	T_ExchgParam.T_StationCommon.xOnlineValueModified_St1:=fbCompareProfileProcessValue.xProcessValueModified;
END_ACTION
ACTION ResetVisu:
(* waiting for reset *)
	RisingEdgeReset(CLK:=T_Visu.T_CtrleVisu.xReset);
	IF RisingEdgeReset.Q THEN
		(* call functionblock init. *)
		fbQvisInitPage(	T_Visu:=T_Visu);
		T_Visu.T_CtrleVisu.xDone:=FALSE;
		T_Visu.T_CtrleVisu.iFunction:=0;
		T_Visu.T_CtrleVisu.xErr:=FALSE;
		T_Visu.T_CtrleVisu.udiErrorID:=0;
		T_Visu.T_PlcParam.dwSetNewPage:=0;
		T_Visu.T_PlcParam.dwActualPage:=0;
		T_Visu.T_PlcParam.dwPreviousPage:=0;
		T_ExchgParam.T_Visu.iQVisActivNewPage:=0;
		T_ExchgParam.T_TeachIn.iSetup_AxisSel:=1;
		T_ExchgParam.T_StationCommon.xBlockSelectAutoMode:=FALSE;
		InitSavePages;
		awSaveStateTaskBar[0]:=awSaveStateTaskBar[1]:=awSaveStateTaskBar[2]:=awSaveStateTaskBar[3]:=awSaveStateTaskBar[4]:=1;
		iSaveSetupMode:=1;
		(* Activ reset structure control action *)
		T_Visu.T_CtrleAction.xReset:=TRUE;
		(* Activ reset structure control process *)
		T_Visu.T_CtrleProcess.xReset:=TRUE;
		RisingEdgeReseTProcess(CLK:=FALSE);
		(* active confirmation *)
		xConfirmResetFB:=TRUE;
		(* exit function bloc *)
		RETURN;
	ELSE
		IF xConfirmResetFB THEN
			(* confirm reset FB *)
			T_Visu.T_CtrleVisu.xDone:=TRUE;
			T_Visu.T_CtrleVisu.xErr:=FALSE;
			T_Visu.T_CtrleVisu.udiErrorID:=0;
			(* reset variable *)
			xConfirmResetFB:=FALSE;
			(* activ research if Qvis is activ *)
			xQvisActiv:=TRUE;
			T_Visu.T_CtrleVisu.xQvis:=FALSE;
			dwInCount_QVisCmd:=T_CtrleQVis.dwInCount;
		END_IF
	END_IF;
END_ACTION
ACTION UserLevel:
	RisingEdgeCheckPasswordPage(CLK:=(T_Visu.T_PlcParam.dwActualPage = gT_PageNumber.iAutoMode_UserLevel));
	IF RisingEdgeCheckPasswordPage.Q OR xChangeRandomValue THEN
		xChangeRandomValue:=FALSE;
		(* Der Counter respektive Random muss 9 Stellig sein welches aus dem Zyklusticker der CPU ausgelesen wird *)
		fbGetCpuAccount;
		FBPassword_SystemLevel(	dwCounterHI:= fbGetCpuAccount.cpuCntHiDW,
								dwCounterLOW:=fbGetCpuAccount.cpuCntLoDW);
		T_ExchgParam.T_Visu.T_Level.diRandom:=FBPassword_SystemLevel.diRandom;
	END_IF;
(* Monitor password divers level *)
	(* set Standard Level *)
	RisingEdgeStandardLevel(CLK:=(T_ExchgParam.T_Visu.T_Level.iActLevel = 0));
	IF RisingEdgeStandardLevel.Q THEN
		xChangeRandomValue:=TRUE;
		T_ExchgParam.T_Visu.T_Message.iState:=31;			(* Info: Sie sind nun als Standard angemeldet *)
	END_IF;
	(* set Operator Level *)
	IF T_ExchgParam.T_Visu.T_Level.diPwOperator <> -1 THEN
		IF T_ExchgParam.T_Visu.T_Level.diPwOperator = T_ExchgParam.T_Visu.T_Level.diPwOperatorSaved THEN
		(* pw correct *)
			T_ExchgParam.T_Visu.T_Level.iActLevel:=1;
			T_ExchgParam.T_Visu.T_Message.iState:=1;			(* Info: Sie sind nun als Operator angemeldet *)
		(* wrong pw *)
		ELSE 	T_ExchgParam.T_Visu.T_Message.iState:=204;	(* Warnung: Falsches Operator Passwort *) END_IF
		T_ExchgParam.T_Visu.T_Level.diPwOperator:=-1;
		xChangeRandomValue:=TRUE;
	END_IF;
	(* set system level *)
	IF T_ExchgParam.T_Visu.T_Level.diPwSystem <> -1 THEN
		IF T_ExchgParam.T_Visu.T_Level.diPwSystem = FBPassword_SystemLevel.diPwSystem THEN
		(* pw correct *)
			T_ExchgParam.T_Visu.T_Level.iActLevel:=2;
			T_ExchgParam.T_Visu.T_Message.iState:=2;			(* Info: Sie sind nun als System angemeldet *)
		(* wrong pw *)
		ELSE 	T_ExchgParam.T_Visu.T_Message.iState:=205; 		(* Warnung: Falsches System Passwort *) END_IF
		T_ExchgParam.T_Visu.T_Level.diPwSystem:=-1;
		xChangeRandomValue:=TRUE;
	END_IF

	IF (T_ExchgParam.T_Visu.T_Level.iActLevel > 1) THEN
		T_ExchgParam.T_StationCommon.xSystemLevelActive:=TRUE;
	ELSE
		T_ExchgParam.T_StationCommon.xSystemLevelActive:=FALSE;
	END_IF;
END_ACTION
ACTION VisuFunction_Axis:
	xTmp:=	xAxisStop OR xAxisStopAll OR xAxisTogglePower OR
			xAxisReset OR xAxisMoveContinous OR xAxisMoveAbsolut OR
			xAxisMoveRelative OR xAxisTeachPosition;

	T_ExchgParam.T_TeachIn.xDisableAxisSelectButton:=xTmp;	(* Auswahl der Achsen muss gesperrt werden im Fall einer Aktiven VisuFunktion für Achsen *)

	IF IxJoystick_X_Plus THEN
		T_ExchgParam.T_TeachIn.xJogInc_Common_Setup_Axis:=TRUE;
		T_ExchgParam.T_Visu.T_Message.iState:=35;	(* Info: Achsen auf Jog Bewegung gesetzt ! *)
	END_IF;
	IF IxJoystick_X_Minus THEN
		T_ExchgParam.T_TeachIn.xJogInc_Common_Setup_Axis:=FALSE;
		T_ExchgParam.T_Visu.T_Message.iState:=34;	(* Info: Achsen auf Ink Bewegung gesetzt ! *)
	END_IF;

(* Bewegung einer Achse stoppen *)
	IF xAxisStop THEN
		(* Step stop axis *)
		CASE iStepAction OF
		(* check Ressource *)
		1:	xTmp:=	TRUE;
			IF xTmp THEN
				(* next Step *)
				iStepAction :=10;
				xStepActionDone:=FALSE;
			(* activ error *)
			ELSE
				iStepAction:=95;
			END_IF
			xAxisMoveContinous:=FALSE;
		(* stop axis *)
		10:	ptrTCommonAxis^.T_CtrleSingle.iFunction:=5;
			ptrTCommonAxis^.T_CtrleSingle.xExecute:=TRUE;
			(* next step *)
			iStepAction:=20;
			xStepActionDone:=FALSE;
		(* waiting stop confirmation *)
		20:	IF NOT(xStepActionDone) THEN
			(* release execution *)
				ptrTCommonAxis^.T_CtrleSingle.xExecute:=FALSE;
				(* confirm step *)
				xStepActionDone:=TRUE;
			ELSE
				IF ptrTCommonAxis^.T_CtrleSingle.xDone THEN
				(* next step *)
					iStepAction:=90;
					xStepActionDone:=FALSE;
					T_ExchgParam.T_Visu.T_Message.iState:=277;	(* Warnung: Achse wurde gestoppt ! *)
				END_IF
			END_IF
		(* action done *)
		90:	T_Visu.T_CtrleAction.xDone:=TRUE;
			T_Visu.T_CtrleAction.xNotReady:=FALSE;
			T_Visu.T_CtrleAction.xErr:=FALSE;
			T_Visu.T_CtrleAction.udiErrorID:=0;
			xAxisStop:=FALSE;
		(* axis not ready *)
		95:	TimerNotReady(IN:=TRUE);
			xAxisStop:=FALSE;
		END_CASE
	END_IF;

(* Bewegung aller Achse stoppen *)
	IF xAxisStopAll THEN
		(* Step stop axis *)
		CASE iStepAction OF
		(* check Ressource *)
		1:	xTmp:=	TRUE;
			IF xTmp THEN
				(* next Step *)
				iStepAction :=10;
				xStepActionDone:=FALSE;
			(* activ error *)
			ELSE
				iStepAction:=95;
			END_IF
			xAxisMoveContinous:=FALSE;
		(* stop axis *)
		10:	IF xAxisStopAll THEN
				ptrTAxisZ_St1^.T_CtrleSingle.iFunction:=5;
				ptrTAxisZ_St1^.T_CtrleSingle.xExecute:=TRUE;
				ptrTAxisS_St1^.T_CtrleSingle.iFunction:=5;
				ptrTAxisS_St1^.T_CtrleSingle.xExecute:=TRUE;
			END_IF;
			(* next step *)
			iStepAction:=20;
			xStepActionDone:=FALSE;
		(* waiting stop confirmation *)
		20:	IF NOT(xStepActionDone) THEN
			(* release execution *)
				(* confirm step *)
				xStepActionDone:=TRUE;
			ELSE
				IF ptrTAxisZ_St1^.T_CtrleSingle.xDone AND ptrTAxisS_St1^.T_CtrleSingle.xDone THEN
				(* next step *)
					iStepAction:=90;
					xStepActionDone:=FALSE;
					T_ExchgParam.T_Visu.T_Message.iState:=277;	(* Warnung: Achse wurde gestoppt ! *)
				END_IF
			END_IF
		(* action done *)
		90:	T_Visu.T_CtrleAction.xDone:=TRUE;
			T_Visu.T_CtrleAction.xNotReady:=FALSE;
			T_Visu.T_CtrleAction.xErr:=FALSE;
			T_Visu.T_CtrleAction.udiErrorID:=0;
			xAxisStopAll:=FALSE;
		(* axis not ready *)
		95:	TimerNotReady(IN:=TRUE);
			xAxisStopAll:=FALSE;
		END_CASE
	END_IF;

(* Achsen Drehmoment Ein/Aus Toggeln *)
	IF xAxisTogglePower THEN
		(* Step toogle axis power *)
		CASE iStepAction OF
		(* check axis *)
		1:	xTmp:=	ptrTCommonAxis^.T_CtrleSingle.xDone
					AND ptrTCommonAxis^.T_CtrleSingle.xNotMoving
					AND NOT(ptrTCommonAxis^.T_CtrleSingle.xErr)
					AND NOT(ptrTCommonAxis^.T_CtrleSingle.xExecute);
			IF xTmp THEN
				iStepAction:=10;
			ELSE
				iStepAction:=95;
			END_IF
		(* activ function axis *)
		10:	IF ptrTCommonAxis^.T_CtrleSingle.xPower THEN ptrTCommonAxis^.T_CtrleSingle.iFunction:=4;
				ELSE ptrTCommonAxis^.T_CtrleSingle.iFunction:=3; END_IF
			ptrTCommonAxis^.T_CtrleSingle.xExecute:=TRUE;
			(* next step *)
			iStepAction:=20;
			xStepActionDone:=FALSE;
		(* confirm execution *)
		20:	IF NOT(xStepActionDone) THEN
			(* confirm execution *)
				ptrTCommonAxis^.T_CtrleSingle.xExecute:=FALSE;
				xStepActionDone:=TRUE;
			ELSE
				IF ptrTCommonAxis^.T_CtrleSingle.xDone THEN
					IF (ptrTCommonAxis^.T_CtrleSingle.iFunction = 3) THEN
						T_ExchgParam.T_Visu.T_Message.iState:=7;	(* Info: Achsenstrom EIN ! *)
					ELSE
						T_ExchgParam.T_Visu.T_Message.iState:=8;	(* Info: Achsenstrom AUS ! *)
					END_IF
				(* confirm action next step *)
					iStepAction:=90;
					xStepActionDone:=FALSE;
				END_IF
			END_IF
		(* action done *)
		90:	T_Visu.T_CtrleAction.xDone:=TRUE;
			T_Visu.T_CtrleAction.xNotReady:=FALSE;
			T_Visu.T_CtrleAction.xErr:=FALSE;
			T_Visu.T_CtrleAction.udiErrorID:=0;
			xAxisTogglePower:=FALSE;
		(* Axis not ready *)
		95:	TimerNotReady(IN:=TRUE);
			xAxisTogglePower:=FALSE;
		END_CASE
	END_IF

(* Achse Resetten *)
	IF xAxisReset THEN
		(* Step reset axis *)
		CASE iStepAction OF
		(* check axis *)
		1:	xTmp:=	NOT(ptrTCommonAxis^.T_CtrleSingle.xExecute);
			IF xTmp THEN
				iStepAction:=10;
			ELSE iStepAction:=95;
			END_IF
		(* activ function axis *)
		10:	ptrTCommonAxis^.T_CtrleSingle.iFunction:=1;
			ptrTCommonAxis^.T_CtrleSingle.xExecute:=TRUE;
			(* next step *)
			iStepAction:=20;
			xStepActionDone:=FALSE;
		(* confirm execution *)
		20:	IF NOT(xStepActionDone) THEN
			(* confirm execution *)
				ptrTCommonAxis^.T_CtrleSingle.xExecute:=FALSE;
				xStepActionDone:=TRUE;
			ELSE
				IF ptrTCommonAxis^.T_CtrleSingle.xDone THEN
					T_ExchgParam.T_Visu.T_Message.iState:=9;	(* Info: Achse erfolgreich Zurückgesetzt ! *)
				(* confirm action next step *)
					iStepAction:=90;
					xStepActionDone:=FALSE;
				END_IF
			END_IF
		(* action done *)
		90:	T_Visu.T_CtrleAction.xDone:=TRUE;
			T_Visu.T_CtrleAction.xNotReady:=FALSE;
			T_Visu.T_CtrleAction.xErr:=FALSE;
			T_Visu.T_CtrleAction.udiErrorID:=0;
			xAxisReset:=FALSE;
		(* Axis not ready *)
		95:	TimerNotReady(IN:=TRUE);
			xAxisReset:=FALSE;
		END_CASE
	END_IF

(* Achse Geschwindigkeitsmodus *)
	IF xAxisMoveContinous THEN
		(* Step move continuous velocity *)
		CASE iStepAction OF
		(* check axis *)
		1:	xTmp:=	ptrTCommonAxisActive^.T_CtrleSingle.xDone
					AND ptrTCommonAxisActive^.T_CtrleSingle.xReady
					AND ptrTCommonAxisActive^.T_CtrleSingle.xNotMoving
					AND NOT(ptrTCommonAxisActive^.T_CtrleSingle.xErr)
					AND NOT(ptrTCommonAxisActive^.T_CtrleSingle.xExecute);
			IF (ptrTCommonAxisActive^.T_CtrleSingle.lrVelocity = 0) THEN
				(* Geschwindigkeit darf nicht 0 sein *)
				iStepAction:=90;
				T_ExchgParam.T_Visu.T_Message.iState:=288;	(* Warnung: Geschwindigkeit muss grösser als 0 sein ! *)
				RETURN;
			END_IF;
			IF xTmp THEN
				iStepAction:=10;
			ELSE
				iStepAction:=95;
			END_IF
		(* activ function axis *)
		10:	ptrTCommonAxisActive^.T_CtrleSingle.iFunction:=6;
			ptrTCommonAxisActive^.T_CtrleSingle.xExecute:=TRUE;
			ptrTCommonAxisActive^.T_CtrleSingle.lrAcceleration:=TCommonTeachParameter.rAcceleration;
			ptrTCommonAxisActive^.T_CtrleSingle.lrDecceleration:=TCommonTeachParameter.rDeceleration;
			ptrTCommonAxisActive^.T_CtrleSingle.lrJerk:=TCommonTeachParameter.rJerk;
			(* next step *)
			iStepAction:=20;
			xStepActionDone:=FALSE;
			T_ExchgParam.T_Visu.T_Message.iState:=14;	(* Info: Achsenbewegung gestartet ! *)
		(* confirm execution *)
		20:	IF NOT(xStepActionDone) THEN
			(* confirm execution *)
				ptrTCommonAxisActive^.T_CtrleSingle.xExecute:=FALSE;
				xStepActionDone:=TRUE;
			ELSE
				IF ptrTCommonAxisActive^.T_CtrleSingle.xDone THEN
					xStepActionDone:=FALSE;
					(* confirm action next step *)
					iStepAction:=90;
				END_IF
			END_IF
		(* action done *)
		90:	T_Visu.T_CtrleAction.xDone:=TRUE;
			T_Visu.T_CtrleAction.xNotReady:=FALSE;
			T_Visu.T_CtrleAction.xErr:=FALSE;
			T_Visu.T_CtrleAction.udiErrorID:=0;
			xAxisMoveContinous:=FALSE;
		(* axis not ready *)
		95:	TimerNotReady(IN:=TRUE);
			xAxisMoveContinous:=FALSE;
		END_CASE
	END_IF

(* Achse Absolute Positionsbewegung *)
	IF xAxisMoveAbsolut THEN
		(* Step move abs position *)
		CASE iStepAction OF
		(* check axis *)
		1:	xTmp:=	ptrTCommonAxis^.T_CtrleSingle.xDone
					AND ptrTCommonAxis^.T_CtrleSingle.xReady
					AND ptrTCommonAxis^.T_CtrleSingle.xNotMoving
					AND NOT(ptrTCommonAxis^.T_CtrleSingle.xErr)
					AND NOT(ptrTCommonAxis^.T_CtrleSingle.xExecute);
			IF xTmp THEN
				IF NOT(ptrTCommonAxis^.T_CtrleSingle.xRef) THEN
					T_ExchgParam.T_Visu.T_Message.iState:=206;	(* Warnung: Ausgewählte Achse ist nicht referenziert ! *)
					iStepAction:=90;
				ELSE
					iStepAction:=10;
				END_IF
			ELSE
				iStepAction:=95;
			END_IF;
		(* waiting confirmation *)
		10:	(* init. acc/dec/jerk *)
			ptrTCommonAxis^.T_CtrleSingle.lrAcceleration:=TCommonTeachParameter.rAcceleration;
			ptrTCommonAxis^.T_CtrleSingle.lrDecceleration:=TCommonTeachParameter.rDeceleration;
			ptrTCommonAxis^.T_CtrleSingle.lrJerk:=TCommonTeachParameter.rJerk;
			ptrTCommonAxis^.T_CtrleSingle.lrVelocity:=TCommonTeachParameter.rPositionSpeed;
			ptrTCommonAxis^.T_CtrleSingle.lrPosition:=TCommonTeachParameter.rRefPosition;
			ptrTCommonAxis^.T_CtrleSingle.xExecute:=TRUE;
			ptrTCommonAxis^.T_CtrleSingle.iFunction:=7;
			iStepAction:=20;
			xStepActionDone:=FALSE;
			IF NOT(xAxisLimitSwitchActive) THEN
				T_ExchgParam.T_Visu.T_Message.iState:=15;	(* Info: Achse fährt auf ausgewählte Position ! *)
			END_IF;
			gxAxisAbsolutMovementActive:=TRUE;	(* Damit die Achsen mit dem Override gesetzt werden bezüglich der Absoluten Bewegung *)
		(* confirm execution *)
		20:	IF NOT(xStepActionDone) THEN
			(* confirm execution *)
				ptrTCommonAxis^.T_CtrleSingle.xExecute:=FALSE;
				xStepActionDone:=TRUE;
			ELSE
				IF ptrTCommonAxis^.T_CtrleSingle.xDone THEN
					xStepActionDone:=FALSE;
					(* confirm action next step *)
					iStepAction:=90;
					IF NOT(xAxisLimitSwitchActive) THEN
						T_ExchgParam.T_Visu.T_Message.iState:=16;	(* Info: Achsenposition erreicht ! *)
					END_IF;
				END_IF
			END_IF;
		(* action done *)
		90:	T_Visu.T_CtrleAction.xDone:=TRUE;
			T_Visu.T_CtrleAction.xNotReady:=FALSE;
			T_Visu.T_CtrleAction.xErr:=FALSE;
			T_Visu.T_CtrleAction.udiErrorID:=0;
			xAxisMoveAbsolut:=FALSE;
		(* axis not ready *)
		95:	TimerNotReady(IN:=TRUE);
			xAxisMoveAbsolut:=FALSE;
		END_CASE
	END_IF

(* Achse Relative Positionsbewegung *)
	IF xAxisMoveRelative THEN
		(* Step move abs position *)
		CASE iStepAction OF
		(* check axis *)
		1:	xTmp:=	ptrTCommonAxisActive^.T_CtrleSingle.xDone
					AND ptrTCommonAxisActive^.T_CtrleSingle.xReady
					AND ptrTCommonAxisActive^.T_CtrleSingle.xNotMoving
					AND NOT(ptrTCommonAxisActive^.T_CtrleSingle.xErr)
					AND NOT(ptrTCommonAxisActive^.T_CtrleSingle.xExecute);
			IF xTmp THEN
				iStepAction:=10;
			ELSE
				iStepAction:=95;
			END_IF;
		(* Überprüfe Software Endschalter *)
		10:	IF ptrTCommonAxisActive^.T_CtrleSingle.xSWLimitSwitchPosActivated THEN
				IF ((ptrTCommonAxisActive^.T_LiveValue.lrActualPosition + ptrTCommonAxisActive^.T_CtrleSingle.lrDistance) > 0.1) THEN
					(* Überschreibe den Inkrement, damit die Achse nicht einen Fehler auswertet! Melde es dann als Softwareendschalter *)
					ptrTCommonAxisActive^.T_CtrleSingle.lrDistance:=0.09 - ptrTCommonAxisActive^.T_LiveValue.lrActualPosition;
					IF ((ptrTCommonAxisActive^.T_LiveValue.lrActualPosition + 0.01) >= 0.1) THEN
						ptrTCommonAxisActive^.T_CtrleSingle.lrDistance:=0.0;
					END_IF;
				END_IF;
			END_IF;
			iStepAction:=20;
		(* waiting confirmation *)
		20:	(* init. acc/dec/jerk *)
			ptrTCommonAxisActive^.T_CtrleSingle.lrAcceleration:=TCommonTeachParameter.rAcceleration;
			ptrTCommonAxisActive^.T_CtrleSingle.lrDecceleration:=TCommonTeachParameter.rDeceleration;
			ptrTCommonAxisActive^.T_CtrleSingle.lrJerk:=TCommonTeachParameter.rJerk;
			ptrTCommonAxisActive^.T_CtrleSingle.iFunction:=8;	(* Relative Bewegung *)
			ptrTCommonAxisActive^.T_CtrleSingle.xExecute:=TRUE;
			iStepAction:=30;
			xStepActionDone:=FALSE;
			IF NOT(xAxisLimitSwitchActive) THEN
				T_ExchgParam.T_Visu.T_Message.iState:=21;	(* Info: Achse relative Bewegung gestartet ! *)
			END_IF;
		(* confirm execution *)
		30:	IF NOT(xStepActionDone) THEN
			(* confirm execution *)
				ptrTCommonAxisActive^.T_CtrleSingle.xExecute:=FALSE;
				xStepActionDone:=TRUE;
			ELSE
				IF ptrTCommonAxisActive^.T_CtrleSingle.xDone THEN
					xStepActionDone:=FALSE;
					(* confirm action next step *)
					iStepAction:=90;
					IF NOT(xAxisLimitSwitchActive) THEN
						T_ExchgParam.T_Visu.T_Message.iState:=22;	(* Info: Achse relative Bewegung durchgeführt ! *)
					END_IF;
				END_IF
			END_IF;
		(* action done *)
		90:	T_Visu.T_CtrleAction.xDone:=TRUE;
			T_Visu.T_CtrleAction.xNotReady:=FALSE;
			T_Visu.T_CtrleAction.xErr:=FALSE;
			T_Visu.T_CtrleAction.udiErrorID:=0;
			xAxisMoveRelative:=FALSE;
		(* axis not ready *)
		95:	TimerNotReady(IN:=TRUE);
			xAxisMoveRelative:=FALSE;
		END_CASE
	END_IF

(* Z Achse auf WzWechsel Pos oder auf Z Achse auf LadePos setzen *)
	IF xZAxisMoveToToolChangePos OR xZAxisMoveToLoadPos THEN
		(* Step move abs position *)
		CASE iStepAction OF
		(* check axis *)
		1:	xTmp:=	ptrTCommonAxisActive^.T_CtrleSingle.xDone
					AND ptrTCommonAxisActive^.T_CtrleSingle.xReady
					AND ptrTCommonAxisActive^.T_CtrleSingle.xNotMoving
					AND NOT(ptrTCommonAxisActive^.T_CtrleSingle.xErr)
					AND NOT(ptrTCommonAxisActive^.T_CtrleSingle.xExecute);
			IF xTmp THEN
				IF NOT(ptrTCommonAxisActive^.T_CtrleSingle.xRef) THEN
					T_ExchgParam.T_Visu.T_Message.iState:=206;	(* Warnung: Ausgewählte Achse ist nicht referenziert ! *)
					iStepAction:=90;
				ELSE
					iStepAction:=5;
					T_ExchgParam.T_Visu.T_Message.iState:=109;	(* Aufforderung: Z Achse Position anfahren <Enter>, abbrechen <Esc> ? *)
				END_IF
			ELSE
				iStepAction:=95;
			END_IF;
		(* Set Value *)
		5:	IF RisingEdgeKeyPanel_Enter.Q THEN
				(* Display message *)
				tTimeOutAction:=T#999999s;
				iStepAction:=10;
			ELSE
				IF RisingEdgeKeyPanel_Esc.Q THEN
					iStepAction:=90;
					T_ExchgParam.T_Visu.T_Message.iState:=202;	(* Warnung: Aktion abgebrochen ! *)
				END_IF
			END_IF
			(* An other message has been displayed *)
			IF (T_ExchgParam.T_Visu.T_Message.iState<>3) AND (T_ExchgParam.T_Visu.T_Message.iState<>109) AND (T_ExchgParam.T_Visu.T_Message.iState<>202) THEN iStepAction:=90; END_IF
		(* waiting confirmation *)
		10:	(* init. acc/dec/jerk *)
			ptrTCommonAxisActive^.T_CtrleSingle.xExecute:=TRUE;
			ptrTCommonAxisActive^.T_CtrleSingle.iFunction:=7;
			ptrTCommonAxisActive^.T_CtrleSingle.lrPosition:=rZAxisSelectPosition;
			iStepAction:=20;
			xStepActionDone:=FALSE;
			IF NOT(xAxisLimitSwitchActive) THEN
				T_ExchgParam.T_Visu.T_Message.iState:=15;	(* Info: Achse fährt auf ausgewählte Position ! *)
			END_IF;
			gxAxisAbsolutMovementActive:=TRUE;	(* Damit die Achsen mit dem Override gesetzt werden bezüglich der Absoluten Bewegung *)
		(* confirm execution *)
		20:	IF NOT(xStepActionDone) THEN
			(* confirm execution *)
				ptrTCommonAxisActive^.T_CtrleSingle.xExecute:=FALSE;
				xStepActionDone:=TRUE;
			ELSE
				IF ptrTCommonAxisActive^.T_CtrleSingle.xDone THEN
					xStepActionDone:=FALSE;
					(* confirm action next step *)
					iStepAction:=90;
					IF NOT(xAxisLimitSwitchActive) THEN
						T_ExchgParam.T_Visu.T_Message.iState:=16;	(* Info: Achsenposition erreicht ! *)
					END_IF;
				END_IF
			END_IF;
		(* action done *)
		90:	T_Visu.T_CtrleAction.xDone:=TRUE;
			T_Visu.T_CtrleAction.xNotReady:=FALSE;
			T_Visu.T_CtrleAction.xErr:=FALSE;
			T_Visu.T_CtrleAction.udiErrorID:=0;
			xZAxisMoveToToolChangePos:=xZAxisMoveToLoadPos:=FALSE;
		(* axis not ready *)
		95:	TimerNotReady(IN:=TRUE);
			xZAxisMoveToToolChangePos:=xZAxisMoveToLoadPos:=FALSE;
		END_CASE
	END_IF

(* Meldung ausgeben, falls bei den Achse Z  Endschalter angefahren werden *)
	IF T_StartUp.T_State.xCompleted THEN
		IF ptrTAxisZ_St1^.T_CtrleSingle.xHWLimitNeg THEN
			T_ExchgParam.T_Visu.T_Message.iState:=209;	(* Warnung: Z-Achse negativer HW Endschalter angefahren ! *)
		END_IF;
		IF ptrTAxisZ_St1^.T_CtrleSingle.xHWLimitPos THEN
			T_ExchgParam.T_Visu.T_Message.iState:=210;	(* Warnung: Z-Achse positiver HW Endschalter angefahren ! *)
		END_IF;
	END_IF;

	IF (T_ExchgParam.T_Visu.T_Message.iState >= 209) AND (T_ExchgParam.T_Visu.T_Message.iState <= 210) THEN
		xAxisLimitSwitchActive:=TRUE;
	ELSE
		xAxisLimitSwitchActive:=FALSE;
	END_IF;

(* Löschen der berechnete Wert für Wippe des Drehmoment Detection *)
IF xResetRockerValue THEN
	grRockerQualityMin:=grRockerQuality;
	grRockerQualityMax:=grRockerQuality;
	grRockerAmplitudeMin:=grRockerAmplitude;
	grRockerAmplitudeMax:=grRockerAmplitude;
	T_ExchgParam.T_StationCommon.rRockerQuality:=grRockerQuality:=0.0;
	T_ExchgParam.T_StationCommon.rRockerAmplitude:=grRockerAmplitude:=0.0;
	T_ExchgParam.T_StationCommon.diRockerCountHC:=gdiRockerCountHC:=0;
	T_ExchgParam.T_StationCommon.diRockerCountHCTime:=gdiRockerCountHCTime:=0;
	T_Visu.T_CtrleAction.xDone:=TRUE;
	T_Visu.T_CtrleAction.xNotReady:=FALSE;
	T_Visu.T_CtrleAction.xErr:=FALSE;
	T_Visu.T_CtrleAction.udiErrorID:=0;
	xResetRockerValue:=FALSE;
END_IF;
END_ACTION
ACTION VisuFunction_AxisTeach:
(* Achse Teach Position *)
	IF xAxisTeachPosition THEN
		CASE iStepAction OF
		(* check axis *)
		1:	xTmp:=	ptrTCommonAxis^.T_CtrleSingle.xDone
					AND ptrTCommonAxis^.T_CtrleSingle.xReady
					AND ptrTCommonAxis^.T_CtrleSingle.xNotMoving
					AND NOT(ptrTCommonAxis^.T_CtrleSingle.xErr)
					AND NOT(ptrTCommonAxis^.T_CtrleSingle.xExecute);
			xReferenceState:=ptrTCommonAxis^.T_CtrleSingle.xRef;
			IF xTmp OR gxHardwareOFF OR gxAxisOFF THEN
				IF NOT(xReferenceState) AND NOT(gxHardwareOFF) AND NOT(gxAxisOFF) THEN
					T_ExchgParam.T_Visu.T_Message.iState:=206;	(* Warnung: Ausgewählte Achse ist nicht referenziert ! *)
					iStepAction:=90;
				ELSE
					iStepAction:=2;
				END_IF
			ELSE
				iStepAction:=95;
			END_IF;
		(* Überprüfe zuerst ob die ausgewählte Position teach bar ist *)
		2:	 T_ExchgParam.T_Visu.T_Message.iState:=0;
			CASE T_ExchgParam.T_TeachIn.iSetup_AxisSel  OF
			1:	(* Z Axis *)
				IF NOT(T_NovRam.T_Parameter.T_StationWork[1].T_StProcess.xConfigActive) THEN
					IF (T_ExchgParam.T_TeachIn.arAxis[T_ExchgParam.T_TeachIn.iSetup_AxisSel].iTeachSelPos = 0) THEN
						T_ExchgParam.T_Visu.T_Message.iState:=207;			(* Warnung: Neue Position kann nicht versetzt werden ! *)
					ELSIF (T_ExchgParam.T_TeachIn.arAxis[T_ExchgParam.T_TeachIn.iSetup_AxisSel].iTeachSelPos = 6) THEN
						T_ExchgParam.T_Visu.T_Message.iState:=208;			(* Warnung: Ausgewählte Position kann nicht gespeichert werden ! *)
					END_IF;
				ELSE
					IF (T_ExchgParam.T_TeachIn.arAxis[T_ExchgParam.T_TeachIn.iSetup_AxisSel].iTeachSelPos = 0) THEN
						T_ExchgParam.T_Visu.T_Message.iState:=207;			(* Warnung: Neue Position kann nicht versetzt werden ! *)
					ELSIF (T_ExchgParam.T_TeachIn.arAxis[T_ExchgParam.T_TeachIn.iSetup_AxisSel].iTeachSelPos <= 4) THEN
						T_ExchgParam.T_Visu.T_Message.iState:=208;			(* Warnung: Ausgewählte Position kann nicht gespeichert werden ! *)
					ELSIF (T_ExchgParam.T_TeachIn.arAxis[T_ExchgParam.T_TeachIn.iSetup_AxisSel].iTeachSelPos = 6) THEN
						T_ExchgParam.T_Visu.T_Message.iState:=208;			(* Warnung: Ausgewählte Position kann nicht gespeichert werden ! *)
					END_IF;
				END_IF;
			END_CASE
			IF (T_ExchgParam.T_Visu.T_Message.iState = 0) THEN
				iStepAction:=10;
			ELSE
				(* Action has been cancelled *)
				iStepAction:=90;
			END_IF;
		(* Display message to ask for confirmation *)
		10:	T_ExchgParam.T_Visu.T_Message.iState:=103;	(* Aufforderung: Speichern bestätigen <Enter>, abbrechen <Esc> ? *)
			iStepAction:=20;
		(* waiting for key <Enter> or <Esc> *)
		20:	IF RisingEdgeKeyPanel_Enter.Q THEN
					iStepAction:=30;
			ELSIF RisingEdgeKeyPanel_Esc.Q THEN
					 iStepAction:=90;
					T_ExchgParam.T_Visu.T_Message.iState:=202;	(* Warnung: Aktion abgebrochen ! *)
			 END_IF
			(* An other message has been displayed *)
			IF (T_ExchgParam.T_Visu.T_Message.iState<>103) AND (T_ExchgParam.T_Visu.T_Message.iState<>202) THEN iStepAction:=90; END_IF
		30:	T_ExchgParam.T_Visu.T_Message.iState:=0;
			(*copy actual value to tmp variable*)
			rtmpAxisPosZ:=LREAL_TO_REAL(TStation_Work_St1.THWWorkStation.TAxisZ.T_LiveValue.lrActualPosition);
			CASE T_ExchgParam.T_TeachIn.iSetup_AxisSel  OF
			1:	(* Z Axis *)
				CASE T_ExchgParam.T_TeachIn.arAxis[T_ExchgParam.T_TeachIn.iSetup_AxisSel].iTeachSelPos OF
				(* < Z LadePos > *)
				1:	T_NovRam.T_Parameter.T_StationWork[gciStationSt1].T_StProcess.rPositionLoad:=rtmpAxisPosZ;
				(* < Z Bearb StartPos > *)
				2:	T_NovRam.T_Parameter.T_StationWork[gciStationSt1].T_StProcess.rPositionStartProc:=rtmpAxisPosZ;
				(* < Z ZentrierPos > *)
				3:	T_NovRam.T_Parameter.T_StationWork[gciStationSt1].T_StProcess.rCentringPosZ1Axis:=rtmpAxisPosZ;
				(* < Z Bearb EndPos > *)
				4:	T_NovRam.T_Parameter.T_StationWork[gciStationSt1].T_StProcess.rPositionEndProc:=rtmpAxisPosZ;
				(* < Z WzWechsel Pos > *)
				5:	T_NovRam.T_Parameter.T_StationWork[gciStationSt1].T_StProcess.rPositionToolChange:=rtmpAxisPosZ;
				(* < Z Bearb EndPos berechn. > *)
				7:	garPositionEndProcCalc[1]:=rtmpAxisPosZ;
					T_ExchgParam.T_StationCommon.rPositionEndProcCalc:=rtmpAxisPosZ;
				(* < Z Bearb EndPos Max > *)
				8:	T_NovRam.T_Parameter.T_StationWork[gciStationSt1].T_StProcess.rPositionEndProcMaxInc:=rtmpAxisPosZ;
				(* < Z ZentrierPos berechn. > *)
				9:	garCentringEndProcCalc[1]:=rtmpAxisPosZ;
					T_ExchgParam.T_StationCommon.rCentringEndProcCalc:=rtmpAxisPosZ;
				(* < Z WzZylinder Pos > *)
				10:	T_NovRam.T_Parameter.T_StationWork[gciStationSt1].T_StProcess.rZPositionCylindricalArea:=rtmpAxisPosZ;
				END_CASE;
				xUpdateStationParameter:=TRUE;
			END_CASE;
			(* Speichern der Daten in den NovRAM *)
			iStepAction:=70;
		70:	IF (garPositionEndProcCalc[1] <> T_ExchgParam.T_StationCommon.rPositionEndProcCalc) THEN
				T_ExchgParam.T_StationCommon.rPositionEndProcCalc:=garPositionEndProcCalc[1];
			END_IF;
			IF (garCentringEndProcCalc[1] <> T_ExchgParam.T_StationCommon.rCentringEndProcCalc) THEN
				T_ExchgParam.T_StationCommon.rCentringEndProcCalc:=garCentringEndProcCalc[1];
			END_IF;
			xAction_SaveNovRAM:=TRUE;
			xBlockSetNovRamAction_End:=TRUE;
			iStepActionNovRam:=1;
			iStepAction:=80;
		80:	IF NOT(xAction_SaveNovRAM) THEN
				iStepAction:=90;
				T_ExchgParam.T_Visu.T_Message.iState:=25;	(* Info: Ausgewählte Position ist nun gespeichert ! *)
			END_IF;
		(* axis not ready *)
		95:	TimerNotReady(IN:=TRUE);
			xAxisTeachPosition:=FALSE;
		(* slow/fast configuration done *)
		90:	T_Visu.T_CtrleAction.xDone:=TRUE;
			T_Visu.T_CtrleAction.xNotReady:=FALSE;
			T_Visu.T_CtrleAction.xErr:=FALSE;
			T_Visu.T_CtrleAction.udiErrorID:=0;
			xAxisTeachPosition:=FALSE;
		END_CASE
	END_IF
END_ACTION
ACTION VisuFunction_ChangePassword:
(* Ändern des Operator Passwortes *)
	IF xChangeOperatorPassword THEN
		CASE iStepAction OF
		(* Display message to ask for confirmation *)
		1:	T_ExchgParam.T_Visu.T_Level.xShow_Overlay_NewPassword:=TRUE;
			T_ExchgParam.T_Visu.T_Level.diInputOldPasword:=0;
			T_ExchgParam.T_Visu.T_Level.diInputNewPasword:=0;
			T_ExchgParam.T_Visu.T_Level.diInputRepeatPasword:=0;
			T_ExchgParam.T_Visu.T_Level.xButton_OK:=FALSE;
			T_ExchgParam.T_Visu.T_Level.xButton_Abord:=FALSE;
			iStepAction:=10;
		10:	IF T_ExchgParam.T_Visu.T_Level.xButton_OK THEN
				T_ExchgParam.T_Visu.T_Level.xButton_OK:=FALSE;
				 tTimeOutAction:=TimerAction.ET+T#3s;
				iStepAction:=20;
			END_IF;
			IF T_ExchgParam.T_Visu.T_Level.xButton_Abord THEN
				T_ExchgParam.T_Visu.T_Level.xButton_Abord:=FALSE;
				iStepAction:=90;
			END_IF;
			IF TimerAction.Q THEN iStepAction:=90; END_IF;
		(* Überprüfe Eingabe des alten Passwort *)
		20:	IF (T_ExchgParam.T_Visu.T_Level.diInputOldPasword = T_ExchgParam.T_Visu.T_Level.diPwOperatorSaved) THEN
				(* Eingabe Korrekt *)
				iStepAction:=30;
			ELSE
				T_ExchgParam.T_Visu.T_Message.iState:=214;	(* Warnung: Altes Operator Passwort falsch eingegeben ! *)
				iStepAction:=90;
			END_IF;
		(* Überprüfe Eingabe des neuen Passwort mit der Eingabe des bestätigten neuen Passwortes *)
		30:	IF (T_ExchgParam.T_Visu.T_Level.diInputNewPasword = T_ExchgParam.T_Visu.T_Level.diInputRepeatPasword) THEN
				(* Eingabe Korrekt *)
				iStepAction:=40;
			ELSE
				T_ExchgParam.T_Visu.T_Message.iState:=215;	(* Warnung: Keine Übereinstimmung der beiden neuen Operator Passwörter ! *)
				iStepAction:=90;
			END_IF;
		(* Speichern des neuen Passwortes *)
		40:	T_Password.T_Ctrle.udiSetOperatorPassword:=T_ExchgParam.T_Visu.T_Level.diInputNewPasword;
			T_Password.T_Ctrle.xExecute:=TRUE;
			T_Password.T_Ctrle.iFunction:=2;
			(* next Step *)
			iStepAction :=50;
			xStepActionDone:=FALSE;
		(* wait save confirmation *)
		50:	IF NOT(xStepActionDone) THEN
				T_Password.T_Ctrle.xExecute:=FALSE;
				(* Überschreiben des alten Passwortes *)
				T_ExchgParam.T_Visu.T_Level.diPwOperatorSaved:=T_ExchgParam.T_Visu.T_Level.diInputNewPasword;
				(* confirm Step *)
				xStepActionDone:=TRUE;
			ELSE
				IF T_Password.T_Ctrle.xDone THEN
				(* next Step *)
					iStepAction :=90;
					xStepActionDone:=FALSE;
					T_ExchgParam.T_Visu.T_Message.iState:=36;	(* Info: Neues Operator Passwort wurde gespeichert und ist Aktiv ! *)
				ELSE	IF T_Password.T_Ctrle.xErr THEN
							iStepAction:=99;
							xStepActionDone:=FALSE;
						END_IF
				END_IF
			END_IF
		(* save done *)
		90:	T_Visu.T_CtrleAction.xDone:=TRUE;
			T_Visu.T_CtrleAction.xNotReady:=FALSE;
			T_Visu.T_CtrleAction.xErr:=FALSE;
			T_Visu.T_CtrleAction.udiErrorID:=0;
			xChangeOperatorPassword:=FALSE;
			T_ExchgParam.T_Visu.T_Level.xShow_Overlay_NewPassword:=FALSE;
		(* error *)
		99:	T_Visu.T_CtrleAction.xDone:=FALSE;
			T_Visu.T_CtrleAction.xNotReady:=FALSE;
			T_Visu.T_CtrleAction.xErr:=TRUE;
			T_Visu.T_CtrleAction.udiErrorID:=16#F1000 + T_Password.T_Ctrle.iFunction;
			xChangeOperatorPassword:=FALSE;
			T_ExchgParam.T_Visu.T_Level.xShow_Overlay_NewPassword:=FALSE;
			T_Password.T_Ctrle.xReset:=TRUE;
		END_CASE
	ELSE
		T_ExchgParam.T_Visu.T_Level.xShow_Overlay_NewPassword:=FALSE;
	END_IF
END_ACTION
ACTION VisuFunction_CylinderValve:
(* Set cylinder analog value *)
	IF xCylSetServoAnalogValue THEN
		(* Step analog Wert *)
		CASE iStepAction OF
		(* check cylinder state *)
		1:	xTmp:=	ptrTCommonCylinderValve^.T_CtrleCyl.xDone
					AND NOT(ptrTCommonCylinderValve^.T_CtrleCyl.xExecute)
					AND NOT(ptrTCommonCylinderValve^.T_CtrleCyl.xErr);
			(* next step *)
			IF xTmp THEN iStepAction:=10; ELSE iStepAction:=95; END_IF
		(* activ function set analog value *)
		10:	ptrTCommonCylinderValve^.T_CtrleCyl.iFunction:=4;
			ptrTCommonCylinderValve^.T_CtrleCyl.xExecute:=TRUE;
			(* next step *)
			iStepAction:=20;
			xStepActionDone:=FALSE;
		(* wait confirmation *)
		20:	IF NOT(xStepActionDone) THEN
			(* release execution *)
				ptrTCommonCylinderValve^.T_CtrleCyl.xExecute:=FALSE;
				xStepActionDone:=TRUE;
			ELSE
				IF ptrTCommonCylinderValve^.T_CtrleCyl.xDone THEN
				(* action done *)
					iStepAction:=90;
					xStepActionDone:=FALSE;
					T_ExchgParam.T_Visu.T_Message.iState:=37;	(* Info: Kraft wurde gesetzt ! *)
				END_IF
			END_IF
		(* action done *)
		90:	T_Visu.T_CtrleAction.xDone:=TRUE;
			T_Visu.T_CtrleAction.xNotReady:=FALSE;
			T_Visu.T_CtrleAction.xErr:=FALSE;
			T_Visu.T_CtrleAction.udiErrorID:=0;
			xCylSetServoAnalogValue:=FALSE;
		(* cylinder not ready *)
		95:	TimerNotReady(IN:=TRUE);
			xCylSetServoAnalogValue:=FALSE;
		END_CASE
	END_IF;

(* Zylinder/Ventile Ein/Aus Toggeln *)
	IF xCylValveToggleOnOff THEN
		(* Step toggle Zustand *)
		CASE iStepAction OF
		(* check cylinder state *)
		1:	xTmp:=	ptrTCommonCylinderValve^.T_CtrleCyl.xDone
					AND NOT(ptrTCommonCylinderValve^.T_CtrleCyl.xExecute)
					AND NOT(ptrTCommonCylinderValve^.T_CtrleCyl.xErr);
			(* next step *)
			IF xTmp THEN iStepAction:=10; ELSE iStepAction:=95; END_IF
		(* toggle cylinder state *)
		10:	ptrTCommonCylinderValve^.T_CtrleCyl.iFunction:=51;
			ptrTCommonCylinderValve^.T_CtrleCyl.xExecute:=TRUE;
			IF (ptrTCommonCylinderValve^.iCylinderTpye = 1) THEN
				ptrTCommonCylinderValve^.T_CtrleCyl.T_Analog.rForceIn:=T_NovRAM.T_Parameter.T_StationWork[gciStationSt1].T_OnlineChange.rForceDeflection;
			END_IF;
			IF (ptrTCommonCylinderValve^.iCylinderTpye = 2) THEN
				ptrTCommonCylinderValve^.T_CtrleCyl.T_Analog.rForceIn:=T_NovRAM.T_Parameter.T_StationWork[gciStationSt1].T_OnlineChange.rTorqueLevelHC;
			END_IF;
			IF (ptrTCommonCylinderValve^.iCylinderTpye = 3) THEN
				ptrTCommonCylinderValve^.T_CtrleCyl.T_Analog.rForceIn:=T_NovRAM.T_Parameter.T_StationWork[gciStationSt1].T_StProcess.rTorqueLevel_Overload;
				TStation_Work_St1.THWWorkStation.TCylToolTorqueHC.T_CtrleCyl.T_Analog.rForceIn:=T_NovRAM.T_Parameter.T_StationWork[gciStationSt1].T_OnlineChange.rTorqueLevelHC;
			END_IF;
			(* next step *)
			iStepAction:=20;
			xStepActionDone:=FALSE;
		(* wait confirmation *)
		20:	IF NOT(xStepActionDone) THEN
			(* release execution *)
				ptrTCommonCylinderValve^.T_CtrleCyl.xExecute:=FALSE;
				xStepActionDone:=TRUE;
			ELSE
				IF ptrTCommonCylinderValve^.T_CtrleCyl.xDone THEN
				(* action done *)
					iStepAction:=90;
					xStepActionDone:=FALSE;
					T_ExchgParam.T_Visu.T_Message.iState:=38;	(* Info: Zustand des Zylinderausganges wurde gewechselt ! *)
				END_IF
			END_IF
		(* action done *)
		90:	T_Visu.T_CtrleAction.xDone:=TRUE;
			T_Visu.T_CtrleAction.xNotReady:=FALSE;
			T_Visu.T_CtrleAction.xErr:=FALSE;
			T_Visu.T_CtrleAction.udiErrorID:=0;
			xCylValveToggleOnOff:=FALSE;
		(* cylinder not ready *)
		95:	TimerNotReady(IN:=TRUE);
			xCylValveToggleOnOff:=FALSE;
		END_CASE
	END_IF;

(* Zylinder Drucklos schalten *)
	IF xCylPressurelessON THEN
		(* Step toggle Zustand *)
		CASE iStepAction OF
		(* check cylinder state *)
		1:	xTmp:=	ptrTCommonCylinderValve^.T_CtrleCyl.xDone
					AND NOT(ptrTCommonCylinderValve^.T_CtrleCyl.xExecute)
					AND NOT(ptrTCommonCylinderValve^.T_CtrleCyl.xErr);
			(* next step *)
			IF xTmp THEN iStepAction:=10; ELSE iStepAction:=95; END_IF
		(* toggle cylinder state *)
		10:	ptrTCommonCylinderValve^.T_CtrleCyl.xReset:=TRUE;	(* Drucklos setzen *)
			(* next step *)
			iStepAction:=20;
			xStepActionDone:=FALSE;
		(* wait confirmation *)
		20:	IF NOT(xStepActionDone) THEN
			(* release execution *)
				ptrTCommonCylinderValve^.T_CtrleCyl.xReset:=FALSE;
				xStepActionDone:=TRUE;
			ELSE
				IF ptrTCommonCylinderValve^.T_CtrleCyl.xDone THEN
				(* action done *)
					iStepAction:=90;
					xStepActionDone:=FALSE;
					T_ExchgParam.T_Visu.T_Message.iState:=73;	(* Info: Zylinder ist Drucklos geschaltet ! *)
				END_IF
			END_IF
		(* action done *)
		90:	T_Visu.T_CtrleAction.xDone:=TRUE;
			T_Visu.T_CtrleAction.xNotReady:=FALSE;
			T_Visu.T_CtrleAction.xErr:=FALSE;
			T_Visu.T_CtrleAction.udiErrorID:=0;
			xCylPressurelessON:=FALSE;
		(* cylinder not ready *)
		95:	TimerNotReady(IN:=TRUE);
			xCylPressurelessON:=FALSE;
		END_CASE
	END_IF;

(* Zyl WzDrehmoment oder WzDrehmomentÜberlast EIN/AUS *)
	IF xCylTorqueOnOff OR xCylTorqueOverloadOnOff THEN
		(* Step toggle Zustand *)
		IF xCylTorqueOnOff THEN
			ptrTCommonCylinderValveTmp:=ADR(TStation_Work_St1.THWWorkStation.TCylToolTorqueHC);
		ELSE
			ptrTCommonCylinderValveTmp:=ADR(TStation_Work_St1.THWWorkStation.TCylToolTorqueOverload);
		END_IF;
		CASE iStepAction OF
		(* check cylinder state *)
		1:	xTmp:=	ptrTCommonCylinderValveTmp^.T_CtrleCyl.xDone
					AND NOT(ptrTCommonCylinderValveTmp^.T_CtrleCyl.xExecute)
					AND NOT(ptrTCommonCylinderValveTmp^.T_CtrleCyl.xErr);
			(* next step *)
			IF xTmp THEN iStepAction:=10; ELSE iStepAction:=95; END_IF
		(* toggle cylinder state *)
		10:	ptrTCommonCylinderValveTmp^.T_CtrleCyl.iFunction:=51;
			ptrTCommonCylinderValveTmp^.T_CtrleCyl.xExecute:=TRUE;
			IF (ptrTCommonCylinderValveTmp^.iCylinderTpye = 2) THEN
				ptrTCommonCylinderValveTmp^.T_CtrleCyl.T_Analog.rForceIn:=T_NovRAM.T_Parameter.T_StationWork[gciStationSt1].T_OnlineChange.rTorqueLevelHC;
			END_IF;
			IF (ptrTCommonCylinderValveTmp^.iCylinderTpye = 3) THEN
				ptrTCommonCylinderValveTmp^.T_CtrleCyl.T_Analog.rForceIn:=T_NovRAM.T_Parameter.T_StationWork[gciStationSt1].T_StProcess.rTorqueLevel_Overload;
				TStation_Work_St1.THWWorkStation.TCylToolTorqueHC.T_CtrleCyl.T_Analog.rForceIn:=T_NovRAM.T_Parameter.T_StationWork[gciStationSt1].T_OnlineChange.rTorqueLevelHC;
			END_IF;
			(* next step *)
			iStepAction:=20;
			xStepActionDone:=FALSE;
		(* wait confirmation *)
		20:	IF NOT(xStepActionDone) THEN
			(* release execution *)
				ptrTCommonCylinderValveTmp^.T_CtrleCyl.xExecute:=FALSE;
				xStepActionDone:=TRUE;
			ELSE
				IF ptrTCommonCylinderValveTmp^.T_CtrleCyl.xDone THEN
				(* action done *)
					iStepAction:=90;
					xStepActionDone:=FALSE;
					T_ExchgParam.T_Visu.T_Message.iState:=38;	(* Info: Zustand des Zylinderausganges wurde gewechselt ! *)
				END_IF
			END_IF
		(* action done *)
		90:	T_Visu.T_CtrleAction.xDone:=TRUE;
			T_Visu.T_CtrleAction.xNotReady:=FALSE;
			T_Visu.T_CtrleAction.xErr:=FALSE;
			T_Visu.T_CtrleAction.udiErrorID:=0;
			xCylTorqueOnOff:=xCylTorqueOverloadOnOff:=FALSE;
		(* cylinder not ready *)
		95:	TimerNotReady(IN:=TRUE);
			xCylTorqueOnOff:=xCylTorqueOverloadOnOff:=FALSE;
		END_CASE
	END_IF;
END_ACTION
ACTION VisuFunction_ErrorManagement:
(* Löschen der Fehlerliste *)
	IF xDeleteErrorList THEN
		(* Step saving NovRAM *)
		CASE iStepAction OF
		(* check NovRAM *)
		1:	xTmp:=	T_NovRAM.T_Ctrle.xDone
					AND NOT(T_NovRAM.T_Ctrle.xExecute)
					AND NOT(T_NovRAM.T_Ctrle.xErr);
			IF xTmp THEN
				(* next Step *)
				iStepAction :=10;
			(* activ error *)
			ELSE iStepAction:=95; END_IF
		10:	(* For delete the error, it need the system level *)
			IF (T_ExchgParam.T_Visu.T_Level.iActLevel <> 2) THEN
				T_ExchgParam.T_Visu.T_Message.iState:=216;	(* Warnung: Diese Parameter können nur auf SystemLevel geändert werden ! *)
				iStepAction:=90;
				RETURN;
			END_IF;
			T_ExchgParam.T_Visu.T_Message.iState:=103;	(* Aufforderung: Speichern bestätigen <Enter>, abbrechen <Esc> ? *)
			(* next Step *)
			iStepAction :=20;
		(* waiting for saving confirmation key <Enter> or <Esc> *)
		20:	IF RisingEdgeKeyPanel_Enter.Q THEN
			(* Display message *)
				T_ExchgParam.T_Visu.T_Message.iState:=3;	(* Info: Start speichern... *)
				(* next step *)
				iStepAction:=30;
			ELSE
				IF RisingEdgeKeyPanel_Esc.Q THEN
					iStepAction:=90;
					T_ExchgParam.T_Visu.T_Message.iState:=202;	(* Warnung: Aktion abgebrochen ! *)
				END_IF
			END_IF
			(* An other message has been displayed *)
			IF (T_ExchgParam.T_Visu.T_Message.iState<>3) AND (T_ExchgParam.T_Visu.T_Message.iState<>103) AND (T_ExchgParam.T_Visu.T_Message.iState<>202) THEN iStepAction:=90; END_IF
		30:	FOR ii:=1 TO 20 DO
				T_NovRAM.T_Parameter.T_ErrorNrList.adiErrorListMachine[ii]:=0;
				T_NovRAM.T_Parameter.T_ErrorNrList.asErrorTimeStampMachine[ii]:='';
			END_FOR;
			(* activ save *)
			T_NovRAM.T_Ctrle.xExecute:=TRUE;
			T_NovRAM.T_Ctrle.iFunction:=2;
			(* next Step *)
			iStepAction :=40;
			xStepActionDone:=FALSE;
		(* wait save confirmation *)
		40:	IF NOT(xStepActionDone) THEN
				T_NovRAM.T_Ctrle.xExecute:=FALSE;
				(* confirm Step *)
				xStepActionDone:=TRUE;
			ELSE
				IF T_NovRAM.T_Ctrle.xDone THEN
				(* next Step *)
					iStepAction :=90;
					xStepActionDone:=FALSE;
					T_ExchgParam.T_SafetyCtrl.xUpdateErrorList:=TRUE;
					T_ExchgParam.T_Visu.T_Message.iState:=39;	(* Info: Fehlerliste wurde gelöscht ! *)
				END_IF
			END_IF
		(* save done *)
		90:	T_Visu.T_CtrleAction.xDone:=TRUE;
			T_Visu.T_CtrleAction.xNotReady:=FALSE;
			T_Visu.T_CtrleAction.xErr:=FALSE;
			T_Visu.T_CtrleAction.udiErrorID:=0;
			xDeleteErrorList:=FALSE;
		(* NovRAM not ready *)
		95:	TimerNotReady(IN:=TRUE);
			xDeleteErrorList:=FALSE;
		END_CASE;
	END_IF;
(* Quittieren des Fehler/Warnung *)
	IF xResetErrorWarning THEN
		CASE iStepAction OF
		1:	T_ExchgParam.T_SafetyCtrl.xResetErrorWarning:=TRUE;
			iStepAction:=10;
		10:	IF NOT(T_ExchgParam.T_SafetyCtrl.xResetErrorWarning) THEN
				iStepAction:=90;
				T_ExchgParam.T_Visu.T_Message.iState:=41;	(* Info: Fehler wurde quittiert ! *)
			END_IF;
		(* save done *)
		90:	T_Visu.T_CtrleAction.xDone:=TRUE;
			T_Visu.T_CtrleAction.xNotReady:=FALSE;
			T_Visu.T_CtrleAction.xErr:=FALSE;
			T_Visu.T_CtrleAction.udiErrorID:=0;
			xResetErrorWarning:=FALSE;
		95:	TimerNotReady(IN:=TRUE);
			xResetErrorWarning:=FALSE;
		END_CASE;
	END_IF;
(* Meldungsfenster Öffnen *)
	IF xOpenMessageWindow THEN
		CASE iStepAction OF
		1:	IF (T_ExchgParam.T_SafetyCtrl.bStateMessageError=0) AND (T_ExchgParam.T_SafetyCtrl.bStateMessageInfo=0) AND (T_ExchgParam.T_SafetyCtrl.bStateMessageWarning=0) THEN
				iStepAction:=10;
			ELSE
				T_ExchgParam.T_SafetyCtrl.bStateMessagePreWarning:=0;
				iStepAction:=95;
			END_IF;
		10:	T_ExchgParam.T_SafetyCtrl.bStateMessagePreWarning:=1;
			iStepAction:=90;
		(* not ready *)
		95:	TimerNotReady(IN:=TRUE);
			xOpenMessageWindow:=FALSE;
		(* configuration done *)
		90:	T_Visu.T_CtrleAction.xDone:=TRUE;
			T_Visu.T_CtrleAction.xNotReady:=FALSE;
			T_Visu.T_CtrleAction.xErr:=FALSE;
			T_Visu.T_CtrleAction.udiErrorID:=0;
			xOpenMessageWindow:=FALSE;
		END_CASE
	END_IF;
END_ACTION
ACTION VisuFunction_LampTest:
(* LampTest *)
	IF xLampTestOnOff OR xLampTestBlinkOnOff OR xLampTestActive THEN
		(* set new page *)
		CASE iStepAction OF
		(* check ctrle visu *)
		1: 	(* activ next step *)
			iStepAction:=10;
			xStepActionDone:=FALSE;
		(* Set new page *)
		10:	IF xLampTestOnOff THEN
				xBlinkLampAcitve:=FALSE;
				IF (T_ExchgParam.T_LampTest.abLedControlButton[1] = 0) THEN
					T_ExchgParam.T_BtFunctionPanel.wState:=1;
					xLedControlButtonON:=TRUE;
				ELSE
					T_ExchgParam.T_BtFunctionPanel.wState:=0;
					xLedControlButtonOFF:=TRUE;
				END_IF;
				IF (T_ExchgParam.T_LampTest.abLedControlLamp[1] = 0) THEN
					xLedControlLampON:=TRUE;
				ELSE
					xLedControlLampOFF:=TRUE;
				END_IF;
				IF (T_ExchgParam.T_LampTest.abLedSetupLamp[1] = 0) THEN
					xLedSetupLampON:=TRUE;
				ELSE
					xLedSetupLampOFF:=TRUE;
				END_IF;
				IF xLedControlButtonON AND xLedControlLampON AND xLedSetupLampON THEN
					T_ExchgParam.T_Visu.T_Message.iState:=42;	(* Info: Alle Lampen sind EIN ! *)
				ELSE
					T_ExchgParam.T_Visu.T_Message.iState:=43;	(* Info: Alle Lampen sind AUS ! *)
				END_IF;
				iStepAction:=90;
			END_IF;
			IF xLampTestBlinkOnOff THEN
				IF xBlinkLampAcitve THEN
					T_ExchgParam.T_BtFunctionPanel.wState:=0;
					xLedControlButtonOFF:=xLedControlLampOFF:=xLedSetupLampOFF:=TRUE;
					xBlinkLampAcitve:=FALSE;
					T_ExchgParam.T_Visu.T_Message.iState:=43;	(* Info: Alle Lampen sind AUS ! *)
				ELSE
					T_ExchgParam.T_BtFunctionPanel.wState:=2;
					xBlinkLampAcitve:=TRUE;
					T_ExchgParam.T_Visu.T_Message.iState:=44;	(* Info: Alle Lampen blinken ! *)
				END_IF;
				iStepAction:=90;
			END_IF;
			IF xLampTestActive THEN
				FOR ii:=1 TO 18 DO
					sCopyTextLinesLampIOEngl[ii]:='';
					sCopyTextLinesLampNIOEngl[ii]:='';
					sCopyTextLinesLampIO[ii]:='';
					sCopyTextLinesLampNIO[ii]:='';
				END_FOR;
				T_ExchgParam.T_BtFunctionPanel.wState:=4;
				xBlinkLampAcitve:=FALSE;
				iStepCheckLamp:=1;
				iStepCheckLampNumber:=0;
				iPtrText:=1;
				iTmpPtrText:=1;
				iStepAction:=20;
				T_ExchgParam.T_Visu.T_Message.iState:=45;	(* Info: Lampentest wurde aktiviert ! *)
			END_IF;
			(* activ step *)
			xStepActionDone:=FALSE;
		20:	xLedControlButtonOFF:=xLedControlLampOFF:=xLedSetupLampOFF:=TRUE;
			iStepAction:=30;
		30:	IF NOT(xLedControlButtonOFF) AND NOT(xLedControlLampOFF) AND NOT(xLedSetupLampOFF) THEN
				IF (iStepCheckLamp <= 16) THEN
					iStepCheckLampNumber:=iStepCheckLampNumber + 1;
					T_ExchgParam.T_LampTest.xShowSelectIONIOButton:=TRUE;
					T_ExchgParam.T_LampTest.sControlMessage1Engl:=CONCAT('Please check the ',INT_TO_STRING(iStepCheckLampNumber));
					T_ExchgParam.T_LampTest.sControlMessage1Engl:=CONCAT(T_ExchgParam.T_LampTest.sControlMessage1Engl,'. Lamp!');
					T_ExchgParam.T_LampTest.sControlMessage2Engl:='Is the Lamp lighting? Confirm with Yes or No';
					T_ExchgParam.T_LampTest.sControlMessage1:=CONCAT('Bitte überprüfe die ',INT_TO_STRING(iStepCheckLampNumber));
					T_ExchgParam.T_LampTest.sControlMessage1:=CONCAT(T_ExchgParam.T_LampTest.sControlMessage1,'. Lampe!');
					T_ExchgParam.T_LampTest.sControlMessage2:='Leuchtet die Lampe? Bestätige mit Ja oder Nein';
					iStepAction:=40;
				ELSE
					T_ExchgParam.T_LampTest.xShowSelectIONIOButton:=FALSE;
					T_ExchgParam.T_LampTest.xShowLampTestResult:=TRUE;
					iStepAction:=60;
				END_IF;
			END_IF;
		40:	IF (iStepCheckLamp >= 1) AND (iStepCheckLamp <= 7) THEN
				IF (iStepCheckLamp > 5) THEN
					iStepCheckLamp:=iStepCheckLamp + 1;
				ELSE
					T_ExchgParam.T_LampTest.abLedControlButton[iStepCheckLamp]:=bFct_GetLedState(iLampNumber:=iStepCheckLamp);
				END_IF;
			END_IF;
			IF (iStepCheckLamp >= 7) AND (iStepCheckLamp <= 12) THEN
				iStepCheckLamp:=13;
			END_IF;
			IF (iStepCheckLamp >= 13) AND (iStepCheckLamp <= 15) THEN
				T_ExchgParam.T_LampTest.abLedControlLamp[iStepCheckLamp - 12]:=bFct_GetLedState(iLampNumber:=iStepCheckLamp);
			END_IF;
			IF (iStepCheckLamp >= 16) THEN
				IF (iStepCheckLamp = 16) THEN
					T_ExchgParam.T_LampTest.abLedSetupLamp[iStepCheckLamp - 15]:=bFct_GetLedState(iLampNumber:=iStepCheckLamp);
				ELSE
					iStepCheckLamp:=iStepCheckLamp + 1;
				END_IF;
			END_IF;
			iStepAction:=50;
		50:	IF (iStepCheckLamp <= 16) THEN
				IF T_ExchgParam.T_LampTest.xButtonLampIO THEN
					iTmpPtrText:=iTmpPtrText + 1;
					T_ExchgParam.T_LampTest.xButtonLampIO:=FALSE;
					IF ((iStepCheckLampNumber) < 10) THEN
						sLineNumber:=CONCAT('0',INT_TO_STRING(iStepCheckLampNumber));
					ELSE
						sLineNumber:=INT_TO_STRING(iStepCheckLampNumber);
					END_IF;
					sCopyTextLinesLampIOEngl[iTmpPtrText]:=CONCAT(sLineNumber,'. ');
					sCopyTextLinesLampIOEngl[iTmpPtrText]:=CONCAT(sCopyTextLinesLampIOEngl[iTmpPtrText],sFct_GetLampOrderNumberEngl(xLampdefect:=FALSE,iLampNumber:=iStepCheckLamp));
					sCopyTextLinesLampIO[iTmpPtrText]:=CONCAT(sLineNumber,'. ');
					sCopyTextLinesLampIO[iTmpPtrText]:=CONCAT(sCopyTextLinesLampIO[iTmpPtrText],sFct_GetLampOrderNumberGer(xLampdefect:=FALSE,iLampNumber:=iStepCheckLamp));
					iStepCheckLamp:=iStepCheckLamp + 1;
					iStepAction:=20;
				END_IF;
				IF T_ExchgParam.T_LampTest.xButtonLampNIO THEN
					iPtrText:=iPtrText + 1;
					IF ((iStepCheckLampNumber) < 10) THEN
						sLineNumber:=CONCAT('0',INT_TO_STRING(iStepCheckLampNumber));
					ELSE
						sLineNumber:=INT_TO_STRING(iStepCheckLampNumber);
					END_IF;
					sCopyTextLinesLampNIOEngl[iPtrText]:=CONCAT(sLineNumber,'. ');
					sCopyTextLinesLampNIOEngl[iPtrText]:=CONCAT(sCopyTextLinesLampNIOEngl[iPtrText],sFct_GetLampOrderNumberEngl(xLampdefect:=TRUE,iLampNumber:=iStepCheckLamp));
					sCopyTextLinesLampNIO[iPtrText]:=CONCAT(sLineNumber,'. ');
					sCopyTextLinesLampNIO[iPtrText]:=CONCAT(sCopyTextLinesLampNIO[iPtrText],sFct_GetLampOrderNumberGer(xLampdefect:=TRUE,iLampNumber:=iStepCheckLamp));
					T_ExchgParam.T_LampTest.xButtonLampNIO:=FALSE;
					iStepCheckLamp:=iStepCheckLamp + 1;
					iStepAction:=20;
				END_IF;
			ELSE
				iStepCheckLamp:=iStepCheckLamp + 1;
				iStepAction:=20;
			END_IF;
		60:	IF (iPtrText = 1) THEN
				(* Test Erfolgreich *)
				T_ExchgParam.T_LampTest.sTextLinesEngl:=sCopyTextLinesLampIOEngl;
				T_ExchgParam.T_LampTest.sTextLinesEngl[1]:='All lamps are okay!';
				T_ExchgParam.T_LampTest.sTextLines:=sCopyTextLinesLampIO;
				T_ExchgParam.T_LampTest.sTextLines[1]:='Alle Lampen sind okay!';
			ELSE
				(* mindestens eine Lampe defekt *)
				T_ExchgParam.T_LampTest.sTextLinesEngl:=sCopyTextLinesLampNIOEngl;
				T_ExchgParam.T_LampTest.sTextLinesEngl[1]:='Replace the follow lamps:';
				T_ExchgParam.T_LampTest.sTextLines:=sCopyTextLinesLampNIO;
				T_ExchgParam.T_LampTest.sTextLines[1]:='Folgende Lampen müssen ersetzt werden:';
			END_IF;
			iStepAction:=70;
		70:	IF T_ExchgParam.T_LampTest.xButtonOK THEN
				T_ExchgParam.T_LampTest.xButtonOK:=FALSE;
				T_ExchgParam.T_LampTest.xShowSelectIONIOButton:=FALSE;
				T_ExchgParam.T_LampTest.xShowLampTestResult:=FALSE;
				T_ExchgParam.T_BtFunctionPanel.wState:=0;
				iStepAction:=90;
				T_ExchgParam.T_Visu.T_Message.iState:=46;	(* Info: Lampentest wurde beendet ! *)
			END_IF;
		(* override done *)
		90:	T_Visu.T_CtrleAction.xDone:=TRUE;
			T_Visu.T_CtrleAction.xNotReady:=FALSE;
			T_Visu.T_CtrleAction.xErr:=FALSE;
			T_Visu.T_CtrleAction.udiErrorID:=0;
			xLampTestOnOff:=xLampTestBlinkOnOff:=xLampTestActive:=FALSE;
			T_ExchgParam.T_SafetyCtrl.xDeactivateLamp:=FALSE;
		END_CASE
	END_IF

	IF (T_Visu.T_PlcParam.dwActualPage = gT_PageNumber.iAutoMode_LampTest) THEN
		IF ((NOT(TProcess.T_Ctrle.xExecute) AND TProcess.T_Ctrle.xDone AND NOT(TProcess.T_Ctrle.xError))) THEN
			T_ExchgParam.T_SafetyCtrl.xDeactivateLamp:=TRUE;	(* Ausgänge für die Lampen dürfen überschrieben werden *)
		ELSE
			T_ExchgParam.T_SafetyCtrl.xDeactivateLamp:=FALSE;	(* Wenn diese Seite verlassen wird, dann dürfen die Ausgänge nicht mehr überschrieben werden *)
		END_IF;
	ELSE
		T_ExchgParam.T_SafetyCtrl.xDeactivateLamp:=FALSE;	(* Wenn diese Seite verlassen wird, dann dürfen die Ausgänge nicht mehr überschrieben werden *)
	END_IF;

	IF (T_ExchgParam.T_Visu.xKey_Escape) AND (T_Visu.T_PlcParam.dwActualPage = gT_PageNumber.iAutoMode_LampTest) AND xLampTestActive THEN
		xLedControlButtonOFF:=xLedControlLampOFF:=xLedSetupLampOFF:=TRUE;
		T_ExchgParam.T_LampTest.xShowSelectIONIOButton:=FALSE;
		T_ExchgParam.T_LampTest.xShowLampTestResult:=FALSE;
		T_ExchgParam.T_LampTest.xButtonOK:=FALSE;
		T_ExchgParam.T_LampTest.xButtonLampIO:=FALSE;
		T_ExchgParam.T_LampTest.xButtonLampNIO:=FALSE;
		T_ExchgParam.T_BtFunctionPanel.wState:=0;
		T_Visu.T_CtrleAction.xDone:=TRUE;
		T_Visu.T_CtrleAction.xNotReady:=FALSE;
		T_Visu.T_CtrleAction.xErr:=FALSE;
		T_Visu.T_CtrleAction.udiErrorID:=0;
		xLampTestOnOff:=xLampTestBlinkOnOff:=xLampTestActive:=FALSE;
	END_IF;

	RisingEdgeCheckLampTestPage(CLK:=T_Visu.T_PlcParam.dwActualPage <> gT_PageNumber.iAutoMode_LampTest);
	RisingEdgeCheckLampTestPage1(CLK:=T_Visu.T_PlcParam.dwActualPage = gT_PageNumber.iAutoMode_LampTest);
	IF RisingEdgeCheckLampTestPage.Q OR RisingEdgeCheckLampTestPage1.Q THEN
		xLedControlButtonOFF:=xLedControlLampOFF:=xLedSetupLampOFF:=TRUE;
		xBlinkLampAcitve:=FALSE;
		T_ExchgParam.T_LampTest.xShowSelectIONIOButton:=FALSE;
		T_ExchgParam.T_LampTest.xShowLampTestResult:=FALSE;
		T_ExchgParam.T_LampTest.xButtonOK:=FALSE;
		T_ExchgParam.T_LampTest.xButtonLampIO:=FALSE;
		T_ExchgParam.T_LampTest.xButtonLampNIO:=FALSE;
		T_ExchgParam.T_BtFunctionPanel.wState:=0;
		xLampTestOnOff:=xLampTestBlinkOnOff:=xLampTestActive:=FALSE;
	END_IF;

	IF xBlinkLampAcitve THEN
		CASE iStepBlinkLampActive OF
		1:	TONWaitChangeState(IN:=FALSE);
			xLedControlButtonON:=xLedControlLampON:=xLedSetupLampON:=TRUE;
			iStepBlinkLampActive:=iStepBlinkLampActive + 1;
		2:	TONWaitChangeState(IN:=TRUE,PT:=T#0.5s);
			IF TONWaitChangeState.Q THEN
				TONWaitChangeState(IN:=FALSE);
				xLedControlButtonOFF:=xLedControlLampOFF:=xLedSetupLampOFF:=TRUE;
				iStepBlinkLampActive:=iStepBlinkLampActive + 1;
			END_IF;
		3:	TONWaitChangeState(IN:=TRUE,PT:=T#0.5s);
			IF TONWaitChangeState.Q THEN
				TONWaitChangeState(IN:=FALSE);
				iStepBlinkLampActive:=1;
			END_IF;
		END_CASE;
	ELSE
		TONWaitChangeState(IN:=FALSE);
		iStepBlinkLampActive:=1;
	END_IF;

	IF xLedControlButtonON THEN
		T_ExchgParam.T_LampTest.abLedControlButton[1]:=bFct_GetLedState(iLampNumber:=1);
		T_ExchgParam.T_LampTest.abLedControlButton[2]:=bFct_GetLedState(iLampNumber:=2);
		T_ExchgParam.T_LampTest.abLedControlButton[3]:=bFct_GetLedState(iLampNumber:=3);
		T_ExchgParam.T_LampTest.abLedControlButton[4]:=bFct_GetLedState(iLampNumber:=4);
		T_ExchgParam.T_LampTest.abLedControlButton[5]:=bFct_GetLedState(iLampNumber:=5);
		xLedControlButtonON:=FALSE;
	END_IF;
	IF xLedControlButtonOFF THEN
		T_ExchgParam.T_LampTest.abLedControlButton[1]:=0;
		T_ExchgParam.T_LampTest.abLedControlButton[2]:=0;
		T_ExchgParam.T_LampTest.abLedControlButton[3]:=0;
		T_ExchgParam.T_LampTest.abLedControlButton[4]:=0;
		T_ExchgParam.T_LampTest.abLedControlButton[5]:=0;
		xLedControlButtonOFF:=FALSE;
	END_IF;
	IF xLedControlLampON THEN
		T_ExchgParam.T_LampTest.abLedControlLamp[1]:=bFct_GetLedState(iLampNumber:=13);
		T_ExchgParam.T_LampTest.abLedControlLamp[2]:=bFct_GetLedState(iLampNumber:=14);
		T_ExchgParam.T_LampTest.abLedControlLamp[3]:=bFct_GetLedState(iLampNumber:=15);
		xLedControlLampON:=FALSE;
	END_IF;
	IF xLedControlLampOFF THEN
		T_ExchgParam.T_LampTest.abLedControlLamp[1]:=0;
		T_ExchgParam.T_LampTest.abLedControlLamp[2]:=0;
		T_ExchgParam.T_LampTest.abLedControlLamp[3]:=0;
		xLedControlLampOFF:=FALSE;
	END_IF;
	IF xLedSetupLampON THEN
		T_ExchgParam.T_LampTest.abLedSetupLamp[1]:=bFct_GetLedState(iLampNumber:=16);
		xLedSetupLampON:=FALSE;
	END_IF;
	IF xLedSetupLampOFF THEN
		T_ExchgParam.T_LampTest.abLedSetupLamp[1]:=0;
		xLedSetupLampOFF:=FALSE;
	END_IF;

(* Ausgang für Lampen setzen *)
IF T_ExchgParam.T_SafetyCtrl.xDeactivateLamp THEN
	IF (T_ExchgParam.T_LampTest.abLedControlButton[1] <> 0) THEN
		QxCtrlLampStartButton:=TRUE;
	ELSE
		QxCtrlLampStartButton:=FALSE;
	END_IF;
	IF (T_ExchgParam.T_LampTest.abLedControlButton[2] <> 0) THEN
		QxCtrlLampStopButton:=TRUE;
	ELSE
		QxCtrlLampStopButton:=FALSE;
	END_IF;
	IF (T_ExchgParam.T_LampTest.abLedControlButton[3] <> 0) THEN
		QxCtrlLampAxesCurrentOff:=TRUE;
	ELSE
		QxCtrlLampAxesCurrentOff:=FALSE;
	END_IF;
	IF (T_ExchgParam.T_LampTest.abLedControlButton[4] <> 0) THEN
		QxCtrlLampReleaseButton:=TRUE;
	ELSE
		QxCtrlLampReleaseButton:=FALSE;
	END_IF;
	IF (T_ExchgParam.T_LampTest.abLedControlButton[5] <> 0) THEN
		QxSetupModeLamp:=TRUE;
	ELSE
		QxSetupModeLamp:=FALSE;
	END_IF;
	IF (T_ExchgParam.T_LampTest.abLedControlLamp[1] <> 0) THEN
		QxSignalLampGreen:=TRUE;
	ELSE
		QxSignalLampGreen:=FALSE;
	END_IF;
	IF (T_ExchgParam.T_LampTest.abLedControlLamp[2] <> 0) THEN
		QxSignalLampYellow:=TRUE;
	ELSE
		QxSignalLampYellow:=FALSE;
	END_IF;
	IF (T_ExchgParam.T_LampTest.abLedControlLamp[3] <> 0) THEN
		QxSignalLampRed:=TRUE;
	ELSE
		QxSignalLampRed:=FALSE;
	END_IF;
	IF (T_ExchgParam.T_LampTest.abLedSetupLamp[1] <> 0) THEN
		QxMachineLamp:=TRUE;
	ELSE
		QxMachineLamp:=FALSE;
	END_IF;
END_IF;
END_ACTION
ACTION VisuFunction_MachineLamp:
(* MaschinenLampe ON/OFF *)
	RisingEdgeMachineLamp(CLK:=(UDINT_TO_WORD(T_CtrlePanel.udiButton) = 16#8));
	IF RisingEdgeMachineLamp.Q AND T_StartUp.T_State.xCompleted AND (T_Visu.T_PlcParam.dwActualPage <> gT_PageNumber.iAutoMode_LampTest) THEN
		xTmp:=	TMachineLamp.T_CtrleCyl.xFBActiv
				AND TMachineLamp.T_CtrleCyl.xDone
				AND NOT(TMachineLamp.T_CtrleCyl.xExecute);
		IF xTmp THEN
			TMachineLamp.T_CtrleCyl.iFunction:=51;
			TMachineLamp.T_CtrleCyl.xExecute:=TRUE;
			IF NOT(TMachineLamp.T_CtrleCyl.T_Standard.xActivOn) THEN
				T_ExchgParam.T_Visu.T_Message.iState:=61;	(* Info: Maschinenlampe EIN ! *)
			ELSE
				T_ExchgParam.T_Visu.T_Message.iState:=62;	(* Info: Maschinenlampe AUS ! *)
			END_IF;
		END_IF;
	END_IF;
END_ACTION
ACTION VisuFunction_NovRAM:
(* Action Save NovRAM *)
	IF xAction_SaveNovRAM THEN
		(* Step saving NovRAM *)
		CASE iStepActionNovRam OF
		(* check NovRAM *)
		1:	xTmp:=	T_NovRAM.T_Ctrle.xDone
					AND NOT(T_NovRAM.T_Ctrle.xExecute)
					AND NOT(T_NovRAM.T_Ctrle.xErr);
			IF xTmp THEN
				(* next Step *)
				iStepActionNovRam :=10;
				xStepActionDone:=FALSE;
				IF (T_Visu.T_CtrleAction.iFunction = 1001) AND (T_ExchgParam.T_BtParameterList.bMessageParameter <> 0) THEN
					(* Beim speichern der Parameterliste besteht keine Parameterliste oder man hat nicht die berechtigung dazu *)
					IF (T_ExchgParam.T_BtParameterList.bMessageParameter = 1) THEN
						T_ExchgParam.T_Visu.T_Message.iState:=217;	(* Warnung: Mindestens OperatorLevel wird benötigt ! *)
					ELSIF (T_ExchgParam.T_BtParameterList.bMessageParameter = 2) THEN
						T_ExchgParam.T_Visu.T_Message.iState:=216;	(* Warnung: Diese Parameter können nur auf SystemLevel geändert werden ! *)
					ELSE
						T_ExchgParam.T_Visu.T_Message.iState:=273;	(* Kann nicht gespeichert werden, da keine Parameterliste besteht ! *)
					END_IF;
					iStepActionNovRam:=90;
					RETURN;
				END_IF;
				(* Display message *)
				T_ExchgParam.T_Visu.T_Message.iState:=3;	(* Info: Start speichern... *)
			(* activ error *)
			ELSE
				iStepActionNovRam:=95;
			END_IF
		(* copy value *)
		10:	(* Update visu exchange variable, aber nur falls die Parameterliste angewählt ist *)
			xTmp:=	(T_Visu.T_PlcParam.dwActualPage = gT_PageNumber.iAutoMode_Parameter) OR
					(T_Visu.T_PlcParam.dwActualPage = gT_PageNumber.iHandMode_Parameter) OR
					(T_Visu.T_PlcParam.dwActualPage = gT_PageNumber.iWorkStation_Parameter);
			IF xTmp THEN
				T_NovRAM.T_Parameter.T_Machine.T_ParamSystem:=T_ExchgParam.T_StationCommon.T_Param_Machine.T_ParamSystem;
				T_NovRam.T_Parameter.T_StationWork[gciStationSt1]:=T_ExchgParam.T_StationCommon.T_Param_StationWork;
				T_NovRam.T_Parameter.T_StationWork[gciStationSt1].T_ToolCounter:=T_ExchgParam.T_StationCommon.T_ToolCounter_St1;
				T_NovRam.T_Parameter.T_StationWork[gciStationSt1].T_WPCounter:=T_ExchgParam.T_StationCommon.T_WPCounter_St1;
				xUpdateStationParameter:=TRUE;
			END_IF;
			IF (T_Visu.T_PlcParam.dwActualPage = gT_PageNumber.iHandMode_Parameter)  AND (T_ExchgParam.T_BtParameterList.iEditParam = 117) THEN
				garPositionEndProcCalc[1]:=T_ExchgParam.T_StationCommon.rPositionEndProcCalc;
				garCentringEndProcCalc[1]:=T_ExchgParam.T_StationCommon.rCentringEndProcCalc;
			END_IF;
			(* next Step *)
			iStepActionNovRam :=20;
			xStepActionDone:=FALSE;
		(* activ save *)
		20:	IF NOT(gxHardwareOFF) THEN
				T_NovRAM.T_Ctrle.xExecute:=TRUE;
				T_NovRAM.T_Ctrle.iFunction:=2;
			END_IF;
			IF (garPositionEndProcCalc[1] <> T_ExchgParam.T_StationCommon.rPositionEndProcCalc) THEN
				T_ExchgParam.T_StationCommon.rPositionEndProcCalc:=garPositionEndProcCalc[1];
			END_IF;
			IF (garCentringEndProcCalc[1] <> T_ExchgParam.T_StationCommon.rCentringEndProcCalc) THEN
				T_ExchgParam.T_StationCommon.rCentringEndProcCalc:=garCentringEndProcCalc[1];
			END_IF;
			(* next Step *)
			iStepActionNovRam :=30;
			xStepActionDone:=FALSE;
		(* wait save confirmation *)
		30:	IF NOT(xStepActionDone) THEN
				T_NovRAM.T_Ctrle.xExecute:=FALSE;
				(* confirm Step *)
				xStepActionDone:=TRUE;
			ELSE
				IF T_NovRAM.T_Ctrle.xDone THEN
				(* next Step *)
					iStepActionNovRam :=90;
					xStepActionDone:=FALSE;
					IF (T_ExchgParam.T_Visu.T_Message.iState = 3) THEN
						T_ExchgParam.T_Visu.T_Message.iState:=47;	(* Info: Parameter gespeichert ! *)
					END_IF;
				ELSE	IF T_NovRAM.T_Ctrle.xErr THEN
							iStepActionNovRam:=99;
							xStepActionDone:=FALSE;
						END_IF
				END_IF
			END_IF
		(* save done *)
		90:	IF NOT(xBlockSetNovRamAction_End) THEN
				T_Visu.T_CtrleAction.xDone:=TRUE;
				T_Visu.T_CtrleAction.xNotReady:=FALSE;
				T_Visu.T_CtrleAction.xErr:=FALSE;
				T_Visu.T_CtrleAction.udiErrorID:=0;
			END_IF;
			xAction_SaveNovRAM:=FALSE;
		(* NovRAM not ready *)
		95:	TimerNotReady(IN:=TRUE);
			xAction_SaveNovRAM:=FALSE;
		(* error *)
		99:	T_Visu.T_CtrleAction.xDone:=FALSE;
			T_Visu.T_CtrleAction.xNotReady:=FALSE;
			T_Visu.T_CtrleAction.xErr:=TRUE;
			T_Visu.T_CtrleAction.udiErrorID:=16#F0000 + T_Visu.T_CtrleAction.iFunction;
			IF T_HDD.T_Ctrle.xErr THEN T_Visu.T_CtrleAction.udiErrorID:=16#F1000 + T_HDD.T_Ctrle.iFunction; T_HDD.T_Ctrle.xReset:=TRUE; END_IF
			IF T_Profile.T_Ctrle.xErr THEN T_Visu.T_CtrleAction.udiErrorID:=16#F1000 + T_Visu.T_CtrleAction.iFunction; T_Profile.T_Ctrle.xReset:=TRUE; END_IF
			xAction_SaveNovRAM:=FALSE;
		END_CASE
	END_IF
END_ACTION
ACTION VisuFunction_OnlineChange:
(* OnlineChange Parameter Z Achse Bearbeitungsgeschwindigkeit vorwärts +/- *)
	IF xOnlineChange_Z_ForwardSpeedMore OR xOnlineChange_Z_ForwardSpeedLess THEN
		(* Step set override *)
		CASE iStepAction OF
		(* modif value *)
		1:	rTmp:=T_NovRam.T_Parameter.T_StationWork[gciStationSt1].T_OnlineChangeINC.rWorkingSpeedForward;
			IF xOnlineChange_Z_ForwardSpeedLess THEN rTmp:=rTmp *-1; END_IF
			T_NovRam.T_Parameter.T_StationWork[gciStationSt1].T_OnlineChange.rWorkingSpeedForward
				:=T_NovRam.T_Parameter.T_StationWork[gciStationSt1].T_OnlineChange.rWorkingSpeedForward + rTmp;
			IF T_NovRam.T_Parameter.T_StationWork[gciStationSt1].T_OnlineChange.rWorkingSpeedForward
			     > T_Profile.T_Profile_MinMax.T_Max.rWorkingSpeedForward THEN
				T_NovRam.T_Parameter.T_StationWork[gciStationSt1].T_OnlineChange.rWorkingSpeedForward
					:=T_Profile.T_Profile_MinMax.T_Max.rWorkingSpeedForward; END_IF
			IF T_NovRam.T_Parameter.T_StationWork[gciStationSt1].T_OnlineChange.rWorkingSpeedForward
			     < T_Profile.T_Profile_MinMax.T_Min.rWorkingSpeedForward THEN
				T_NovRam.T_Parameter.T_StationWork[gciStationSt1].T_OnlineChange.rWorkingSpeedForward
					:=T_Profile.T_Profile_MinMax.T_Min.rWorkingSpeedForward; END_IF
			iStepAction:=10;
			xStepActionDone:=FALSE;
		(* set new speed while axis is moving *)
		10:	IF NOT ptrActivStation^.THWWorkStation.TAxisZ.T_CtrleSingle.xNotMoving AND NOT ptrActivStation^.TCtrlOnlineChange.xLockChange_Z_WorkSpeedForward THEN
				ptrActivStation^.THWWorkStation.TAxisZ.T_CtrleSingle.lrVelocity:=T_NovRam.T_Parameter.T_StationWork[gciStationSt1].T_OnlineChange.rWorkingSpeedForward;
				ptrActivStation^.THWWorkStation.TAxisZ.T_CtrleSingle.xExecute:=TRUE;
				ptrActivStation^.THWWorkStation.TAxisZ.T_CtrleSingle.iFunction:=12;
				(* next step *)
				iStepAction:=20;
			ELSE
				(* next step *)
				iStepAction:=90;
			END_IF;
			xStepActionDone:=FALSE;
		(* confirm execution *)
		20: IF NOT(xStepActionDone) THEN
				ptrActivStation^.THWWorkStation.TAxisZ.T_CtrleSingle.xExecute:=FALSE;
				(* confirm step *)
				xStepActionDone:=TRUE;
			ELSE
			(* no confirmation will be sended, confirm override *)
				iStepAction:=90;
				xStepActionDone:=FALSE;
				T_ExchgParam.T_Visu.T_Message.iState:=48;	(* Info: OnlineChange Wert gesetzt ! *)
			END_IF
		(* override done *)
		90:	T_Visu.T_CtrleAction.xDone:=TRUE;
			T_Visu.T_CtrleAction.xNotReady:=FALSE;
			T_Visu.T_CtrleAction.xErr:=FALSE;
			T_Visu.T_CtrleAction.udiErrorID:=0;
			xOnlineChange_Z_ForwardSpeedMore:=FALSE;
			xOnlineChange_Z_ForwardSpeedLess:=FALSE;
			xUpdateStationParameter:=TRUE;
		END_CASE
	END_IF

(* OnlineChange Parameter Z Achse Bearbeitungsgeschwindigkeit rückwärts +/- *)
	IF xOnlineChange_Z_BackwardSpeedMore OR xOnlineChange_Z_BackwardSpeedLess THEN
		(* Step set override *)
		CASE iStepAction OF
		(* modif value *)
		1:	rTmp:=T_NovRam.T_Parameter.T_StationWork[gciStationSt1].T_OnlineChangeINC.rWorkingSpeedBackward;
			IF xOnlineChange_Z_BackwardSpeedLess THEN rTmp:=rTmp *-1; END_IF
			T_NovRam.T_Parameter.T_StationWork[gciStationSt1].T_OnlineChange.rWorkingSpeedBackward
				:=T_NovRam.T_Parameter.T_StationWork[gciStationSt1].T_OnlineChange.rWorkingSpeedBackward + rTmp;
			IF T_NovRam.T_Parameter.T_StationWork[gciStationSt1].T_OnlineChange.rWorkingSpeedBackward
			     > T_Profile.T_Profile_MinMax.T_Max.rWorkingSpeedBackward THEN
				T_NovRam.T_Parameter.T_StationWork[gciStationSt1].T_OnlineChange.rWorkingSpeedBackward
					:=T_Profile.T_Profile_MinMax.T_Max.rWorkingSpeedBackward; END_IF
			IF T_NovRam.T_Parameter.T_StationWork[gciStationSt1].T_OnlineChange.rWorkingSpeedBackward
			     < T_Profile.T_Profile_MinMax.T_Min.rWorkingSpeedBackward THEN
				T_NovRam.T_Parameter.T_StationWork[gciStationSt1].T_OnlineChange.rWorkingSpeedBackward
					:=T_Profile.T_Profile_MinMax.T_Min.rWorkingSpeedBackward; END_IF
			iStepAction:=10;
			xStepActionDone:=FALSE;
		(* set new speed while axis is moving *)
		10:	IF NOT ptrActivStation^.THWWorkStation.TAxisZ.T_CtrleSingle.xNotMoving AND NOT ptrActivStation^.TCtrlOnlineChange.xLockChange_Z_WorkSpeedBackward THEN
				ptrActivStation^.THWWorkStation.TAxisZ.T_CtrleSingle.lrVelocity:=T_NovRam.T_Parameter.T_StationWork[gciStationSt1].T_OnlineChange.rWorkingSpeedBackward;
				ptrActivStation^.THWWorkStation.TAxisZ.T_CtrleSingle.xExecute:=TRUE;
				ptrActivStation^.THWWorkStation.TAxisZ.T_CtrleSingle.iFunction:=12;
				(* next step *)
				iStepAction:=20;
			ELSE
				(* next step *)
				iStepAction:=90;
			END_IF;
			xStepActionDone:=FALSE;
		(* confirm execution *)
		20: IF NOT(xStepActionDone) THEN
				ptrActivStation^.THWWorkStation.TAxisZ.T_CtrleSingle.xExecute:=FALSE;
				(* confirm step *)
				xStepActionDone:=TRUE;
			ELSE
			(* no confirmation will be sended, confirm override *)
				iStepAction:=90;
				xStepActionDone:=FALSE;
				T_ExchgParam.T_Visu.T_Message.iState:=48;	(* Info: OnlineChange Wert gesetzt ! *)
			END_IF
		(* override done *)
		90:	T_Visu.T_CtrleAction.xDone:=TRUE;
			T_Visu.T_CtrleAction.xNotReady:=FALSE;
			T_Visu.T_CtrleAction.xErr:=FALSE;
			T_Visu.T_CtrleAction.udiErrorID:=0;
			xOnlineChange_Z_BackwardSpeedMore:=FALSE;
			xOnlineChange_Z_BackwardSpeedLess:=FALSE;
			xUpdateStationParameter:=TRUE;
		END_CASE
	END_IF

(* OnlineChange Parameter Z Achse rückwärts Offset +/- *)
	IF xOnlineChange_Z_BackwardOffsetMore OR xOnlineChange_Z_BackwardOffsetLess THEN
		(* Step set override *)
		CASE iStepAction OF
		(* modif value *)
		1:	rTmp:=T_NovRam.T_Parameter.T_StationWork[gciStationSt1].T_OnlineChangeINC.rWorkingOffsetBackward;
			IF xOnlineChange_Z_BackwardOffsetLess THEN rTmp:=rTmp *-1; END_IF
			T_NovRam.T_Parameter.T_StationWork[gciStationSt1].T_OnlineChange.rWorkingOffsetBackward
				:=T_NovRam.T_Parameter.T_StationWork[gciStationSt1].T_OnlineChange.rWorkingOffsetBackward + rTmp;
			IF T_NovRam.T_Parameter.T_StationWork[gciStationSt1].T_OnlineChange.rWorkingOffsetBackward
			     > T_Profile.T_Profile_MinMax.T_Max.rWorkingOffsetBackward THEN
				T_NovRam.T_Parameter.T_StationWork[gciStationSt1].T_OnlineChange.rWorkingOffsetBackward
					:=T_Profile.T_Profile_MinMax.T_Max.rWorkingOffsetBackward; END_IF
			IF T_NovRam.T_Parameter.T_StationWork[gciStationSt1].T_OnlineChange.rWorkingOffsetBackward
			     < T_Profile.T_Profile_MinMax.T_Min.rWorkingOffsetBackward THEN
				T_NovRam.T_Parameter.T_StationWork[gciStationSt1].T_OnlineChange.rWorkingOffsetBackward
					:=T_Profile.T_Profile_MinMax.T_Min.rWorkingOffsetBackward; END_IF
			iStepAction:=90;
			T_ExchgParam.T_Visu.T_Message.iState:=48;	(* Info: OnlineChange Wert gesetzt ! *)
		(* override done *)
		90:	T_Visu.T_CtrleAction.xDone:=TRUE;
			T_Visu.T_CtrleAction.xNotReady:=FALSE;
			T_Visu.T_CtrleAction.xErr:=FALSE;
			T_Visu.T_CtrleAction.udiErrorID:=0;
			xOnlineChange_Z_BackwardOffsetMore:=FALSE;
			xOnlineChange_Z_BackwardOffsetLess:=FALSE;
			xUpdateStationParameter:=TRUE;
		END_CASE
	END_IF

(* OnlineChange Parameter ToolTorque Drehmoment HC +/- *)
	IF xOnlineChange_TorqueLevelHCMore OR xOnlineChange_TorqueLevelHCLess THEN
		(* Step set override *)
		CASE iStepAction OF
		(* modif value *)
		1:	rTmp:=T_NovRam.T_Parameter.T_StationWork[gciStationSt1].T_OnlineChangeINC.rTorqueLevelHC;
			IF xOnlineChange_TorqueLevelHCLess THEN rTmp:=rTmp *-1; END_IF
			T_NovRam.T_Parameter.T_StationWork[gciStationSt1].T_OnlineChange.rTorqueLevelHC
				:=T_NovRam.T_Parameter.T_StationWork[gciStationSt1].T_OnlineChange.rTorqueLevelHC + rTmp;
			IF T_NovRam.T_Parameter.T_StationWork[gciStationSt1].T_OnlineChange.rTorqueLevelHC
			     > T_Profile.T_Profile_MinMax.T_Max.rTorqueLevelHC THEN
				T_NovRam.T_Parameter.T_StationWork[gciStationSt1].T_OnlineChange.rTorqueLevelHC
					:=T_Profile.T_Profile_MinMax.T_Max.rTorqueLevelHC; END_IF
			IF T_NovRam.T_Parameter.T_StationWork[gciStationSt1].T_OnlineChange.rTorqueLevelHC
			     < T_Profile.T_Profile_MinMax.T_Min.rTorqueLevelHC THEN
				T_NovRam.T_Parameter.T_StationWork[gciStationSt1].T_OnlineChange.rTorqueLevelHC
					:=T_Profile.T_Profile_MinMax.T_Min.rTorqueLevelHC; END_IF
			iStepAction:=10;
		(* set new speed while axis is moving *)
		10:	IF ptrTCylToolTorqueHC_St1^.T_CtrleCyl.xDone AND ptrTCylToolTorqueOverload_St1^.T_CtrleCyl.xDone AND NOT ptrActivStation^.TCtrlOnlineChange.xLockChangeCylToolTorqueLevel THEN
				ptrTCylToolTorqueHC_St1^.T_CtrleCyl.T_Analog.rForceIn:=T_NovRam.T_Parameter.T_StationWork[gciStationSt1].T_OnlineChange.rTorqueLevelHC;
				ptrTCylToolTorqueHC_St1^.T_CtrleCyl.iFunction:=4;
				ptrTCylToolTorqueHC_St1^.T_CtrleCyl.xExecute:=TRUE;
				ptrTCylToolTorqueOverload_St1^.T_CtrleCyl.T_Analog.rForceIn:=T_NovRam.T_Parameter.T_StationWork[gciStationSt1].T_StProcess.rTorqueLevel_Overload;
				ptrTCylToolTorqueOverload_St1^.T_CtrleCyl.iFunction:=4;
				ptrTCylToolTorqueOverload_St1^.T_CtrleCyl.xExecute:=TRUE;
				(* next step *)
				iStepAction:=20;
			ELSE
				(* next step *)
				iStepAction:=90;
			END_IF;
			xStepActionDone:=FALSE;
		(* confirm execution *)
		20: IF NOT(xStepActionDone) THEN
				ptrTCylToolTorqueHC_St1^.T_CtrleCyl.xExecute:=FALSE;
				(* confirm step *)
				xStepActionDone:=TRUE;
			ELSE
			(* no confirmation will be sended, confirm override *)
				IF ptrTCylToolTorqueHC_St1^.T_CtrleCyl.xDone THEN
					iStepAction:=90;
					xStepActionDone:=FALSE;
					T_ExchgParam.T_Visu.T_Message.iState:=48;	(* Info: OnlineChange Wert gesetzt ! *)
				END_IF;
			END_IF
		(* override done *)
		90:	T_Visu.T_CtrleAction.xDone:=TRUE;
			T_Visu.T_CtrleAction.xNotReady:=FALSE;
			T_Visu.T_CtrleAction.xErr:=FALSE;
			T_Visu.T_CtrleAction.udiErrorID:=0;
			xOnlineChange_TorqueLevelHCMore:=FALSE;
			xOnlineChange_TorqueLevelHCLess:=FALSE;
			xUpdateStationParameter:=TRUE;
		END_CASE
	END_IF

(* OnlineChange Parameter ToolDeflection Auslenkkraft +/- *)
	IF xOnlineChange_DeflectionForceMore OR xOnlineChange_DeflectionForceLess THEN
		(* Step set override *)
		CASE iStepAction OF
		(* modif value *)
		1:	rTmp:=T_NovRam.T_Parameter.T_StationWork[gciStationSt1].T_OnlineChangeINC.rForceDeflection;
			IF xOnlineChange_DeflectionForceLess THEN rTmp:=rTmp *-1; END_IF
			T_NovRam.T_Parameter.T_StationWork[gciStationSt1].T_OnlineChange.rForceDeflection
				:=T_NovRam.T_Parameter.T_StationWork[gciStationSt1].T_OnlineChange.rForceDeflection + rTmp;
			IF T_NovRam.T_Parameter.T_StationWork[gciStationSt1].T_OnlineChange.rForceDeflection
			     > T_Profile.T_Profile_MinMax.T_Max.rForceDeflection THEN
				T_NovRam.T_Parameter.T_StationWork[gciStationSt1].T_OnlineChange.rForceDeflection
					:=T_Profile.T_Profile_MinMax.T_Max.rForceDeflection; END_IF
			IF T_NovRam.T_Parameter.T_StationWork[gciStationSt1].T_OnlineChange.rForceDeflection
			     < T_Profile.T_Profile_MinMax.T_Min.rForceDeflection THEN
				T_NovRam.T_Parameter.T_StationWork[gciStationSt1].T_OnlineChange.rForceDeflection
					:=T_Profile.T_Profile_MinMax.T_Min.rForceDeflection; END_IF
			iStepAction:=10;
			xStepActionDone:=FALSE;
		(* set new speed while axis is moving *)
		10:	IF ptrActivStation^.THWWorkStation.TCylToolDeflection.T_CtrleCyl.xDone AND NOT ptrActivStation^.TCtrlOnlineChange.xLockChangeCylToolDeflectionForce THEN
				ptrActivStation^.THWWorkStation.TCylToolDeflection.T_CtrleCyl.T_Analog.rForceIn:=T_NovRam.T_Parameter.T_StationWork[gciStationSt1].T_OnlineChange.rForceDeflection;
				ptrActivStation^.THWWorkStation.TCylToolDeflection.T_CtrleCyl.iFunction:=4;
				ptrActivStation^.THWWorkStation.TCylToolDeflection.T_CtrleCyl.xExecute:=TRUE;
				(* next step *)
				iStepAction:=20;
			ELSE
				(* next step *)
				iStepAction:=90;
			END_IF;
			xStepActionDone:=FALSE;
		(* confirm execution *)
		20: IF NOT(xStepActionDone) THEN
				ptrActivStation^.THWWorkStation.TCylToolDeflection.T_CtrleCyl.xExecute:=FALSE;
				(* confirm step *)
				xStepActionDone:=TRUE;
			ELSE
			(* no confirmation will be sended, confirm override *)
				IF ptrActivStation^.THWWorkStation.TCylToolDeflection.T_CtrleCyl.xDone THEN
					iStepAction:=90;
					xStepActionDone:=FALSE;
					T_ExchgParam.T_Visu.T_Message.iState:=48;	(* Info: OnlineChange Wert gesetzt ! *)
				END_IF;
			END_IF
		(* override done *)
		90:	T_Visu.T_CtrleAction.xDone:=TRUE;
			T_Visu.T_CtrleAction.xNotReady:=FALSE;
			T_Visu.T_CtrleAction.xErr:=FALSE;
			T_Visu.T_CtrleAction.udiErrorID:=0;
			xOnlineChange_DeflectionForceMore:=FALSE;
			xOnlineChange_DeflectionForceLess:=FALSE;
			xUpdateStationParameter:=TRUE;
		END_CASE
	END_IF

(* OnlineChange Parameter S Achse Bearbeitungsgeschwindigkeit +/- *)
	IF xOnlineChange_S_WorkSpeedMore OR xOnlineChange_S_WorkSpeedLess THEN
		(* Step set override *)
		CASE iStepAction OF
		(* modif value *)
		1:	rTmp:=T_NovRam.T_Parameter.T_StationWork[gciStationSt1].T_OnlineChangeINC.rWorkingSpindleSpeed;
			IF xOnlineChange_S_WorkSpeedLess THEN rTmp:=rTmp *-1; END_IF
			T_NovRam.T_Parameter.T_StationWork[gciStationSt1].T_OnlineChange.rWorkingSpindleSpeed
				:=T_NovRam.T_Parameter.T_StationWork[gciStationSt1].T_OnlineChange.rWorkingSpindleSpeed + rTmp;
			IF T_NovRam.T_Parameter.T_StationWork[gciStationSt1].T_OnlineChange.rWorkingSpindleSpeed
			     > T_Profile.T_Profile_MinMax.T_Max.rWorkingSpindleSpeed THEN
				T_NovRam.T_Parameter.T_StationWork[gciStationSt1].T_OnlineChange.rWorkingSpindleSpeed
					:=T_Profile.T_Profile_MinMax.T_Max.rWorkingSpindleSpeed; END_IF
			IF T_NovRam.T_Parameter.T_StationWork[gciStationSt1].T_OnlineChange.rWorkingSpindleSpeed
			     < T_Profile.T_Profile_MinMax.T_Min.rWorkingSpindleSpeed THEN
				T_NovRam.T_Parameter.T_StationWork[gciStationSt1].T_OnlineChange.rWorkingSpindleSpeed
					:=T_Profile.T_Profile_MinMax.T_Min.rWorkingSpindleSpeed; END_IF
			iStepAction:=10;
			xStepActionDone:=FALSE;
		(* set new speed while axis is moving *)
		10:	IF NOT ptrActivStation^.THWWorkStation.TAxisS.T_CtrleSingle.xNotMoving AND NOT ptrActivStation^.TCtrlOnlineChange.xLockChange_S_WorkSpindleSpeed THEN
				ptrActivStation^.THWWorkStation.TAxisS.T_CtrleSingle.lrVelocity:=T_NovRam.T_Parameter.T_StationWork[gciStationSt1].T_OnlineChange.rWorkingSpindleSpeed;
				ptrActivStation^.THWWorkStation.TAxisS.T_CtrleSingle.xExecute:=TRUE;
				ptrActivStation^.THWWorkStation.TAxisS.T_CtrleSingle.iFunction:=12;
				(* next step *)
				iStepAction:=20;
			ELSE
				(* next step *)
				iStepAction:=90;
			END_IF;
			xStepActionDone:=FALSE;
		(* confirm execution *)
		20: IF NOT(xStepActionDone) THEN
				ptrActivStation^.THWWorkStation.TAxisS.T_CtrleSingle.xExecute:=FALSE;
				(* confirm step *)
				xStepActionDone:=TRUE;
			ELSE
			(* no confirmation will be sended, confirm override *)
				iStepAction:=90;
				xStepActionDone:=FALSE;
				T_ExchgParam.T_Visu.T_Message.iState:=48;	(* Info: OnlineChange Wert gesetzt ! *)
			END_IF
		(* override done *)
		90:	T_Visu.T_CtrleAction.xDone:=TRUE;
			T_Visu.T_CtrleAction.xNotReady:=FALSE;
			T_Visu.T_CtrleAction.xErr:=FALSE;
			T_Visu.T_CtrleAction.udiErrorID:=0;
			xOnlineChange_S_WorkSpeedMore:=FALSE;
			xOnlineChange_S_WorkSpeedLess:=FALSE;
			xUpdateStationParameter:=TRUE;
		END_CASE
	END_IF

	(* Max Werte für Online Change Parameter *)
	IF T_StartUp.T_State.xCompleted THEN
		CASE T_ExchgParam.bToolSpindleActive OF
		1:	(* Maxon Spindel *)
			xFctSetOnlineChangeMaxMin(	ptrProfileOnlineChange:=ADR(T_Profile.T_Profile_MinMax),
										rMaxToolSpindleSpeed:=TStation_Work_St1.THWWorkStation.TCtrlWork.rMaxToolSpindleSpeed,
										rMaxForceDeflection:=T_NovRAM.T_Parameter.T_StationWork[gciStationSt1].T_SpindleSystem.rMaxDeflectionForce,
										rMaxTorqueLevel:=T_NovRAM.T_Parameter.T_StationWork[gciStationSt1].T_TorqueSystem.rMaxTorque,
										rMinTorqueLevel:=0.0);
		2:	(* Beckhoff Spindel L *)
			xFctSetOnlineChangeMaxMin(	ptrProfileOnlineChange:=ADR(T_Profile.T_Profile_MinMax),
										rMaxToolSpindleSpeed:=TStation_Work_St1.THWWorkStation.TCtrlWork.rMaxToolSpindleSpeed,
										rMaxForceDeflection:=T_NovRAM.T_Parameter.T_StationWork[gciStationSt1].T_SpindleSystem_L.rMaxDeflectionForce,
										rMaxTorqueLevel:=T_NovRAM.T_Parameter.T_StationWork[gciStationSt1].T_TorqueSystem_L.rMaxTorque,
										rMinTorqueLevel:=0.0);
		3:	(* Beckhoff Spindel M *)
			xFctSetOnlineChangeMaxMin(	ptrProfileOnlineChange:=ADR(T_Profile.T_Profile_MinMax),
										rMaxToolSpindleSpeed:=TStation_Work_St1.THWWorkStation.TCtrlWork.rMaxToolSpindleSpeed,
										rMaxForceDeflection:=T_NovRAM.T_Parameter.T_StationWork[gciStationSt1].T_SpindleSystem_M.rMaxDeflectionForce,
										rMaxTorqueLevel:=T_NovRAM.T_Parameter.T_StationWork[gciStationSt1].T_TorqueSystem_M.rMaxTorque,
										rMinTorqueLevel:=0.0);
		END_CASE;

		T_ExchgParam.T_ProfileCommon.T_OnlineChange.T_Max:=T_Profile.T_Profile_MinMax.T_Max;
		T_ExchgParam.T_ProfileCommon.T_OnlineChange.T_Min:=T_Profile.T_Profile_MinMax.T_Min;
	END_IF;
END_ACTION
ACTION VisuFunction_ProcessFunction:
(* Prozesse die aus der Stationsebene ausgelöst werden *)
	IF xActionProcStation THEN
		(* Step process machine *)
		CASE iStepAction OF
		(* check process state *)
		1:	iProcessFunctNr:=TProcess.T_Ctrle.iFunctNr;
			xTmp:=	(TProcess.T_Ctrle.xRdy AND TProcess.T_Ctrle.xDone AND NOT(TProcess.T_Ctrle.xError));
			(* next step *)
			IF xTmp THEN
				IF NOT(T_NovRam.T_Parameter.T_StationWork[gciStationSt1].T_AxisState.xReferencedZAxis) THEN
					T_ExchgParam.T_Visu.T_Message.iState:=294;	(* Warnung: Z Achse Ersteinrichtung zuerst durchführen ! *)
					iStepAction:=90;
				ELSE
					IF gxInitialStateActivated THEN
						IF (gxCentringActive OR gxOnlyCentringActive) AND NOT(IxCylWPUnfixAtWorkPos_St1) THEN
							T_ExchgParam.T_Visu.T_Message.iState:=211;	(* Warnung: Zentr.Schlitten von Hand auf Bearb.Position setzen ! *)
							iStepAction:=90;
						ELSE
							iStepAction:=10;
						END_IF;
					ELSE
						T_ExchgParam.T_Visu.T_Message.iState:=293;	(* Warnung: Grundstellungsfahrt zuerst ausführen ! *)
						iStepAction:=90;
					END_IF;
				END_IF;
			ELSE
				iStepAction:=95;
			END_IF;
		(* check process number and start process machine *)
		10:	CASE iProcessFunctNr OF
			(* process available *)
			(*	3=HandBetrieb 1 Loch bearbeitung
				4=WstkEntlade Prozedur
			*)
			3:	T_Visu.T_CtrleProcess.iFunction:=2;
				T_Visu.T_CtrleProcess.xExecute:=TRUE;
				iStepAction:=90;
				T_ExchgParam.T_Visu.T_Message.iState:=49;	(* Info: HandBetrieb Prozess gestartet ! *)
			(* unknown process *)
			ELSE	iStepAction:=95;
			END_CASE
			(* next step *)
			xStepActionDone:=FALSE;
		(* action done *)
		90:	T_Visu.T_CtrleAction.xDone:=TRUE;
			T_Visu.T_CtrleAction.xNotReady:=FALSE;
			T_Visu.T_CtrleAction.xErr:=FALSE;
			T_Visu.T_CtrleAction.udiErrorID:=0;
			xActionProcStation:=FALSE;
		(* cylinder not ready *)
		95:	TimerNotReady(IN:=TRUE);
			xActionProcStation:=FALSE;
		END_CASE
	END_IF;

(* Prozesse die aus der Maschinenebene ausgelöst werden *)
	IF xActionProcMachine THEN
		(* Step process machine *)
		CASE iStepAction OF
		(* check process state *)
		1:	iProcessFunctNr:=TProcess.T_Ctrle.iFunctNr;
			xTmp:=	(TProcess.T_Ctrle.xRdy AND TProcess.T_Ctrle.xDone AND NOT(TProcess.T_Ctrle.xError));
			(* next step *)
			IF xTmp THEN
				IF NOT(T_NovRam.T_Parameter.T_StationWork[gciStationSt1].T_AxisState.xReferencedZAxis) THEN
					T_ExchgParam.T_Visu.T_Message.iState:=294;	(* Warnung: Z Achse Ersteinrichtung zuerst durchführen ! *)
					iStepAction:=90;
				ELSE
					IF (iProcessFunctNr = 1) THEN
						iStepAction:=10;
					ELSIF gxInitialStateActivated THEN
						IF (gxCentringActive OR gxOnlyCentringActive) AND NOT(IxCylWPUnfixAtWorkPos_St1) THEN
							T_ExchgParam.T_Visu.T_Message.iState:=211;	(* Warnung: Zentr.Schlitten von Hand auf Bearb.Position setzen ! *)
							iStepAction:=90;
						ELSE
							iStepAction:=10;
						END_IF;
					ELSE
						T_ExchgParam.T_Visu.T_Message.iState:=293;	(* Warnung: Grundstellungsfahrt zuerst ausführen ! *)
						iStepAction:=90;
					END_IF;
				END_IF;
			ELSE
				iStepAction:=95;
			END_IF;
		(* check process number and start process machine *)
		10:	CASE iProcessFunctNr OF
			(* process available *)
			(*	1=Maschinen Referenzierung
				2=Automat 
			*)
			1..2:	T_Visu.T_CtrleProcess.iFunction:=1;
					T_Visu.T_CtrleProcess.xExecute:=TRUE;
				iStepAction:=90;
				IF (iProcessFunctNr = 1) THEN
					T_ExchgParam.T_Visu.T_Message.iState:=50;	(* Info: Modul Referenzierung gestartet ! *)
				ELSIF (iProcessFunctNr = 2) THEN
					T_ExchgParam.T_Visu.T_Message.iState:=51;	(* Info: Automat gestartet ! *)
					T_ExchgParam.T_StationCommon.xBlockSelectAutoMode:=TRUE;
				END_IF;
			(* unknown process *)
			ELSE	iStepAction:=95;
			END_CASE
			(* next step *)
			xStepActionDone:=FALSE;
		(* action done *)
		90:	T_Visu.T_CtrleAction.xDone:=TRUE;
			T_Visu.T_CtrleAction.xNotReady:=FALSE;
			T_Visu.T_CtrleAction.xErr:=FALSE;
			T_Visu.T_CtrleAction.udiErrorID:=0;
			xActionProcMachine:=FALSE;
		(* cylinder not ready *)
		95:	TimerNotReady(IN:=TRUE);
			xActionProcMachine:=FALSE;
		END_CASE
	END_IF;


	IF TProcess.T_Ctrle.xDone AND NOT(TProcess.T_Ctrle.xError) THEN
		T_ExchgParam.T_StationCommon.bActiveStation_St1St2:=0;	(* Automat nicht Aktiv *)
	ELSIF TProcess.T_Ctrle.xError THEN
		T_ExchgParam.T_StationCommon.bActiveStation_St1St2:=2;	(* Automat Fehler *)
	ELSE
		T_ExchgParam.T_StationCommon.bActiveStation_St1St2:=1;	(* Automat Aktiv *)
	END_IF;
END_ACTION
ACTION VisuFunction_ProcessState:
(* Löschen des Prozesszustandspeicher  *)
	IF xDeleteProcessState THEN
		(* Step  function station  *)
		CASE iStepAction OF
		(* Überprüfe zuerst ob mindestens der OperatorLevel gesetzt ist *)
		1:	xTmp:=	TRUE;
			IF (T_ExchgParam.T_Visu.T_Level.iActLevel < 1) AND NOT(gT_SafetyStatus.xSetupOperateModeActive) THEN
				T_ExchgParam.T_Visu.T_Message.iState:=217;	(* Warnung: Mindestens OperatorLevel wird benötigt ! *)
				iStepAction:=90;
			ELSE
				IF xTmp THEN
					iStepAction:=10;
				ELSE
					iStepAction:=95;
				END_IF;
			END_IF;
		(* Display message to ask for confirmation *)
		10:	T_ExchgParam.T_Visu.T_Message.iState:=103;	(* Aufforderung: Speichern bestätigen <Enter>, abbrechen <Esc> ? *)
			iStepAction:=20;
		(* waiting for key <Enter> or <Esc> *)
		20:	IF RisingEdgeKeyPanel_Enter.Q THEN
				tTimeOutAction:=TimerAction.ET+T#600s;
				iStepAction:=30;
				T_ExchgParam.T_Visu.T_Message.iState:=77;	(* Info: Löschvorgang Automatik Prozesszustand gestartet ! *)
				xStepActionDone:=FALSE;
			ELSE
				IF RisingEdgeKeyPanel_Esc.Q THEN
					iStepAction:=90;
					T_ExchgParam.T_Visu.T_Message.iState:=202;	(* Warnung: Aktion abgebrochen ! *)
				END_IF
			END_IF
			(* An other message has been displayed *)
			IF (T_ExchgParam.T_Visu.T_Message.iState<>103) AND (T_ExchgParam.T_Visu.T_Message.iState<>77) AND (T_ExchgParam.T_Visu.T_Message.iState<>202) THEN iStepAction:=90; END_IF
		(* wait confirmation *)
		30:	T_ExchgParam.T_Visu.T_Message.iState:=78;	(* Info: Automatik Prozesszustand gelöscht ! *)
			gxResetDataAnalysis_St1:=TRUE;
			T_NovRam.T_Parameter.T_Machine.T_ParamAutomat.tAutoProcessTime_St1St2:=T#0s;
			T_NovRam.T_Parameter.T_Machine.T_ParamAutomat.iAutoProcessDay_St1St2:=0;
			T_NovRam.T_Parameter.T_Machine.T_ParamAutomat.diNumberPartWorked_St1St2:=0;
			T_ExchgParam.T_StationCommon.T_Param_Machine.T_ParamAutomat.diNumberPartWorked_St1St2:=0;
			(* action done *)
			iStepAction:=90;
		(* action done *)
		90:	T_Visu.T_CtrleAction.xDone:=TRUE;
			T_Visu.T_CtrleAction.xNotReady:=FALSE;
			T_Visu.T_CtrleAction.xErr:=FALSE;
			T_Visu.T_CtrleAction.udiErrorID:=0;
			xDeleteProcessState:=FALSE;
			T_Visu.T_CtrleAction.xFunctionActive:=FALSE;
		(* function not ready *)
		95:	TimerNotReady(IN:=TRUE);
			xDeleteProcessState:=FALSE;
			T_Visu.T_CtrleAction.xFunctionActive:=FALSE;
		END_CASE
	END_IF

	T_ExchgParam.T_PartQuality.diActual_NumberHoleToWork:=T_NovRam.T_Parameter.T_PartAnalysis[gciStationSt1].diActual_NumberHoleToWork;
	T_ExchgParam.T_PartQuality.sFileName:=T_NovRam.T_Parameter.T_PartAnalysis[gciStationSt1].sFileName;
	T_ExchgParam.T_StationCommon.T_Param_StationWork.T_InfoProcess.diWPNumber:=T_ExchgParam.T_PartQuality.diActual_NumberHoleToWork;

(* Endlos Prozess EIN/AUS *)
(* Zentrieren EIN/AUS *)
(* NurZentrieren EIN/AUS *)
(* Suspenstion EIN/AUS *)
(* ZylWPUnfix EIN/AUS *)
	IF xEndlessProcessOnOff OR xCentringONOFF OR xOnlyCentringONOFF OR xSuspensionONOFF OR xCylWPUnfixONOFF THEN
		(* Step  function station  *)
		CASE iStepAction OF
		(* Überprüfe zuerst ob mindestens der OperatorLevel gesetzt ist *)
		1:	xTmp:=	TRUE;
			IF xEndlessProcessOnOff AND (T_ExchgParam.T_Visu.T_Level.iActLevel < 1) THEN
				T_ExchgParam.T_Visu.T_Message.iState:=217;	(* Warnung: Mindestens OperatorLevel wird benötigt ! *)
				iStepAction:=90;
			ELSE
				IF xTmp THEN
					IF xCentringONOFF OR xOnlyCentringONOFF OR xSuspensionONOFF OR xCylWPUnfixONOFF THEN
						iStepAction:=70;
					ELSE
						iStepAction:=10;
					END_IF
				ELSE
					iStepAction:=95;
				END_IF;
			END_IF;
		(* Display message to ask for confirmation *)
		10:	T_ExchgParam.T_Visu.T_Message.iState:=103;	(* Aufforderung: Speichern bestätigen <Enter>, abbrechen <Esc> ? *)
			iStepAction:=20;
		(* waiting for key <Enter> or <Esc> *)
		20:	IF RisingEdgeKeyPanel_Enter.Q THEN
				iStepAction:=30;
				(* Display message *)
				T_ExchgParam.T_Visu.T_Message.iState:=3;	(* Info: Start speichern... *)
			ELSE
				IF RisingEdgeKeyPanel_Esc.Q THEN
					iStepAction:=90;
					T_ExchgParam.T_Visu.T_Message.iState:=202;	(* Warnung: Aktion abgebrochen ! *)
				END_IF
			END_IF
			(* An other message has been displayed *)
			IF (T_ExchgParam.T_Visu.T_Message.iState<>3) AND (T_ExchgParam.T_Visu.T_Message.iState<>103) AND (T_ExchgParam.T_Visu.T_Message.iState<>202) THEN iStepAction:=90; END_IF
		30:	T_NovRam.T_Parameter.T_Machine.xEndlessProcessActive:=NOT(T_NovRam.T_Parameter.T_Machine.xEndlessProcessActive);
			iStepAction:=40;
		40:	xAction_SaveNovRAM:=TRUE;
			xBlockSetNovRamAction_End:=TRUE;
			iStepActionNovRam:=1;
			iStepAction:=50;
		50:	IF NOT xAction_SaveNovRAM THEN
				iStepAction:=90;
				T_ExchgParam.T_Visu.T_Message.iState:=59;	(* Info: Funktion beendet ! *)
			END_IF;



		70:	IF xCentringONOFF THEN
				gxCentringActive:=NOT(gxCentringActive);
				gxOnlyCentringActive:=FALSE;
			ELSIF xOnlyCentringONOFF THEN
				gxCentringActive:=FALSE;
				gxOnlyCentringActive:=NOT(gxOnlyCentringActive);
			ELSIF xSuspensionONOFF THEN
				IF (T_NovRam.T_Parameter.T_StationWork[1].T_StProcess.rSuspensionBubblerSpeed = 0.0) AND (T_NovRam.T_Parameter.T_StationWork[1].T_StProcess.rSuspensionFeederSpeed = 0.0) THEN
					IF NOT(gxSuspensionONOFF) THEN
						T_ExchgParam.T_Visu.T_Message.iState:=212;	(* Warnung: Suspensionsparameter sind beide auf Null gesetzt ! *)
					ELSE
						gxSuspensionONOFF:=FALSE;
					END_IF;
				ELSE
					gxSuspensionONOFF:=NOT(gxSuspensionONOFF);
				END_IF;
			ELSIF xCylWPUnfixONOFF THEN
				IF NOT(IxCylWPUnfixAtWorkPos_St1) THEN
					IF NOT(QxCylWPUnfix_St1) THEN
						T_ExchgParam.T_Visu.T_Message.iState:=211;	(* Warnung: Zentr.Schlitten von Hand auf Bearb.Position setzen ! *)
					ELSE
						QxCylWPUnfix_St1:=FALSE;
					END_IF;
				ELSE
					QxCylWPUnfix_St1:=NOT(QxCylWPUnfix_St1);
				END_IF;
			END_IF
			T_NovRam.T_Parameter.T_Machine.xEndlessProcessActive:=FALSE;
			iStepAction:=90;

		(* action done *)
		90:	T_Visu.T_CtrleAction.xDone:=TRUE;
			T_Visu.T_CtrleAction.xNotReady:=FALSE;
			T_Visu.T_CtrleAction.xErr:=FALSE;
			T_Visu.T_CtrleAction.udiErrorID:=0;
			xEndlessProcessOnOff:=FALSE;
			xCentringONOFF:=xOnlyCentringONOFF:=FALSE;
			xSuspensionONOFF:=FALSE;
			xCylWPUnfixONOFF:=FALSE;
			T_Visu.T_CtrleAction.xFunctionActive:=FALSE;
		(* function not ready *)
		95:	TimerNotReady(IN:=TRUE);
			xEndlessProcessOnOff:=FALSE;
			xCentringONOFF:=xOnlyCentringONOFF:=FALSE;
			xSuspensionONOFF:=FALSE;
			xCylWPUnfixONOFF:=FALSE;
			T_Visu.T_CtrleAction.xFunctionActive:=FALSE;
		END_CASE
	END_IF

	IF gxCentringActive OR gxOnlyCentringActive THEN
		T_ExchgParam.T_StationCommon.xShowSelectCentringProcess:=TRUE;
	ELSE
		T_ExchgParam.T_StationCommon.xShowSelectCentringProcess:=FALSE;
	END_IF;
	RisingEdgeCheckCentringProcess(CLK:=	(T_ExchgParam.T_StationCommon.T_Param_StationWork.T_StProcess.iCentringSelectProcess <> T_NovRam.T_Parameter.T_StationWork[1].T_StProcess.iCentringSelectProcess));
	IF T_StartUp.T_State.xCompleted AND (T_Visu.T_PlcParam.dwActualPage <> gT_PageNumber.iHandMode_Parameter) THEN
		IF RisingEdgeCheckCentringProcess.Q THEN
			T_NovRam.T_Parameter.T_StationWork[1].T_StProcess.iCentringSelectProcess:=T_ExchgParam.T_StationCommon.T_Param_StationWork.T_StProcess.iCentringSelectProcess;
		END_IF;
	END_IF;
END_ACTION
ACTION VisuFunction_ProcessStop:
(* Stoppen vom Prozess welches über den HandBetrieb ausgelöst wurde *)
	IF xProcStationStop THEN
		(* Step  function station stop  *)
		CASE iStepAction OF
		(* Überprüfe zuerst den Zustand des Prozesses ob es überhaupt zulässt, den Prozess zu stoppen *)
		1:	xTmp:=	TProcess.T_Ctrle.xRdy
					AND NOT(TProcess.T_Ctrle.xStop)
					AND NOT(TProcess.T_Ctrle.xDone)
					AND NOT(TProcess.T_Ctrle.xError)
					AND NOT(TProcess.T_Ctrle.xAbordProcess);
			T_Visu.T_CtrleProcess.xReset:=TRUE;
			IF xTmp THEN
				iStepAction:=10;
			(* not ready to execute stop *)
			ELSE iStepAction:=95; END_IF
		10:	TProcess.T_Ctrle.xStop:=TRUE;
			(* next step *)
			iStepAction:=20;
			xStepActionDone:=FALSE;
		(* wait confirmation *)
		20:	T_ExchgParam.T_Visu.T_Message.iState:=232;	(* Warnung: Unverzüglicher Zyklus-Stopp ! *)
			IF NOT(xStepActionDone) THEN
			(* release execution *)
				xStepActionDone:=TRUE;
			ELSE
				(* Warten bis Prozess beendet ist *)
				IF NOT(TProcess.T_Ctrle.xStop) AND TProcess.T_Ctrle.xDone THEN
					(* action done *)
					iStepAction:=30;
					xStepActionDone:=FALSE;
					T_ExchgParam.T_Visu.T_Message.iState:=236;	(* Warnung: Prozess wurde gestoppt ! *)
					T_VisuQVis.T_CtrleVisu.iFunction:=1;
					T_VisuQVis.T_PlcParam.dwSetNewPage:=dwSaveVisuPage;
					T_VisuQVis.T_CtrleVisu.xExecute:=TRUE;
				END_IF;
			END_IF;
		30:	IF NOT(T_VisuQVis.T_CtrleVisu.xExecute) AND T_VisuQVis.T_CtrleVisu.xDone THEN
				iStepAction:=90;
			END_IF;
		(* action done *)
		90:	T_Visu.T_CtrleAction.xDone:=TRUE;
			T_Visu.T_CtrleAction.xNotReady:=FALSE;
			T_Visu.T_CtrleAction.xErr:=FALSE;
			T_Visu.T_CtrleAction.udiErrorID:=0;
			xProcStationStop:=FALSE;
			T_StartUp.T_State.xBlockChangeMovementVisu:=FALSE;
		(* function not ready *)
		95:	TimerNotReady(IN:=TRUE);
			xProcStationStop:=FALSE;
		END_CASE;
	END_IF;

	IF xProcMachineStop THEN
		(* Step  function station stop  *)
		CASE iStepAction OF
		1:	iStepAction:=90;
			IF xProcMachineStop THEN
				iStepActionStop:=1;
				xTmpProcMachineStop:=TRUE;
			END_IF;
		(* action done *)
		90:	T_Visu.T_CtrleAction.xDone:=TRUE;
			T_Visu.T_CtrleAction.xNotReady:=FALSE;
			T_Visu.T_CtrleAction.xErr:=FALSE;
			T_Visu.T_CtrleAction.udiErrorID:=0;
			xProcMachineStop:=FALSE;
		END_CASE;
	END_IF;

(* Stoppen vom Prozess welches über den Automat ausgelöst wurde *)
	IF xTmpProcMachineStop THEN
		(* Step  function station stop  *)
		CASE iStepActionStop OF
		(* Überprüfe zuerst den Zustand des Prozesses ob es überhaupt zulässt, den Prozess zu stoppen *)
		1:	xTmp:=	TProcess.T_Ctrle.xRdy
					AND NOT(TProcess.T_Ctrle.xStop)
					AND NOT(TProcess.T_Ctrle.xDone)
					AND NOT(TProcess.T_Ctrle.xError)
					AND NOT(TProcess.T_Ctrle.xAbordProcess);
			IF xTmp THEN
				iStepActionStop:=10;
			(* not ready to execute stop *)
			ELSE iStepActionStop:=95; END_IF
		10:	TProcess.T_Ctrle.xStop:=TRUE;
			(* next step *)
			iStepActionStop:=20;
			xStepActionDoneStop:=FALSE;
		(* wait confirmation *)
		20:	T_ExchgParam.T_Visu.T_Message.iState:=232;	(* Warnung: Unverzüglicher Zyklus-Stopp ! *)
			IF NOT(xStepActionDoneStop) THEN
			(* release execution *)
				xStepActionDoneStop:=TRUE;
			ELSE
				IF NOT(TProcess.T_Ctrle.xStop) AND TProcess.T_Ctrle.xDone THEN
					(* Für Maschinenreferenzieren und Wstk Entlade Prozess wird der Prozess beendet *)
					xProcessAbordet:=TRUE;
					iStepActionStop:=90;
					xStepActionDoneStop:=FALSE;
					T_ExchgParam.T_Visu.T_Message.iState:=236;	(* Warnung: Prozess wurde gestoppt ! *)
				END_IF;
			END_IF;
		(* action done *)
		90:	xTmpProcMachineStop:=FALSE;
		(* function not ready *)
		95:	xTmpProcMachineStop:=FALSE;
		END_CASE;
	END_IF;
END_ACTION
ACTION VisuFunction_ProfileManagement:
(* Erstmalige Kopiervorgang der Profile *)
	IF xAction_CopyProfileToProcess THEN
		(* Set copy action *)
		CASE iStepAction OF
		(* Set default value *)
		1:	xFctSetDefaultValueStaticProfile(ptrT_DefaultProfileParameter:=ADR(T_Profile.T_DefaultProfileParameter));
			(* Init. display value *)
			xProfileFileNotFoundSt1:=FALSE;
			xWrongProfilNameReadedSt1:=FALSE;
			xProfileFileWrongSyntaxSt1:=FALSE;
			xProfileFileWrongSyntax:=FALSE;
			iStepAction:=2; (* Überprüfe zuerst als nächstes ob das USB Stick ansprechbar ist *)
		(* check first if USB-Stick exist *)
		2:	T_Profile.T_Ctrle.iFunction:=3;	(* check if the USB-Stick exist *)
			T_Profile.T_Ctrle.xExecute:=TRUE;
			iStepAction:=3;
		3:	IF NOT(T_Profile.T_Ctrle.xExecute) AND T_Profile.T_Ctrle.xDone THEN
				(* USB Stick exist *)
				iStepAction:=4;
			END_IF;
			IF NOT(T_Profile.T_Ctrle.xExecute) AND T_Profile.T_Ctrle.xErr THEN
				(* USB-Stick does not exist *)
				T_ExchgParam.T_Visu.T_Message.iState:=0;	(* Meldung zurücksetzen *)
				T_Profile.T_Ctrle.xReset:=TRUE;
				iStepAction:=98;
			END_IF;
		(* Read First all exist Profilname for manage the profile  *)
		4:	T_Profile.T_Ctrle.sPathAndFileName:='PROFILE\';
			T_Profile.T_Ctrle.iFunction:=6;
			T_Profile.T_Ctrle.xExecute:=TRUE;
			iStepAction:=5;
		5:	IF NOT(T_Profile.T_Ctrle.xExecute) AND T_Profile.T_Ctrle.xDone THEN
				(* all readed profile are ok *)
				iStepAction:=10;
			END_IF;
			IF NOT(T_Profile.T_Ctrle.xExecute) AND T_Profile.T_Ctrle.xErr THEN
				(* Wrong Syntax-->1 File of Profile is corrupted *)
				T_ExchgParam.T_Visu.T_Message.iState:=0;	(* Meldung zurücksetzen *)
				T_Profile.T_IDProfileStation[1].iNumber:=1;
				T_Profile.T_IDProfileStation[1].sName:='Default';
				T_Profile.T_Ctrle.xReset:=TRUE;
				xProfileFileWrongSyntax:=TRUE;
				iStepAction:=90;
			END_IF;
		(* activ reading profile file *)
		10:	IF T_NovRam.T_Parameter.T_StationWork[gciStationSt1].T_InfoProcess.iProfile > 0 AND T_NovRam.T_Parameter.T_StationWork[gciStationSt1].T_InfoProcess.iProfile <= csiMaxProfile THEN
				T_Profile.T_Ctrle.sPathAndFileName:='PROFILE\';
				T_Profile.T_Id.iNumber:=T_NovRam.T_Parameter.T_StationWork[gciStationSt1].T_InfoProcess.iProfile;
				T_Profile.T_Id.sName:=T_NovRam.T_Parameter.T_StationWork[gciStationSt1].T_InfoProcess.sProfileName;
				T_Profile.T_Ctrle.iFunction:=4;	(* read the profile file *)
				T_Profile.T_Ctrle.xExecute:=TRUE;
				(* next step *)
				iStepAction:=20;
			ELSE iStepAction:=25; END_IF
		20:	IF NOT T_Profile.T_Ctrle.xExecute AND T_Profile.T_Ctrle.xDone THEN
				(* Setzen des aktuellen Prozessabbild welches vom NovRAM ist *)
				T_Profile.T_LoadProfileParameter:=T_Profile.T_CopyProfileParameter;
				T_ExchgParam.T_StationCommon.T_Param_StationWork.T_InfoProcess.iProfile:=T_NovRam.T_Parameter.T_StationWork[gciStationSt1].T_InfoProcess.iProfile;
				T_ExchgParam.T_StationCommon.T_Param_StationWork.T_InfoProcess.sProfileName:=T_Profile.T_Id.sName;
				garPositionEndProcCalc[gciStationSt1]:=T_NovRam.T_Parameter.arZ1AxisCalcEndPosSaveProfile[gciStationSt1,T_NovRam.T_Parameter.T_StationWork[gciStationSt1].T_InfoProcess.iProfile];
				garCentringEndProcCalc[gciStationSt1]:=T_NovRam.T_Parameter.arZ1CentringCalcEndPosSaveProfile[gciStationSt1,T_NovRam.T_Parameter.T_StationWork[gciStationSt1].T_InfoProcess.iProfile];
				(* check if the read name of the profil file is the same as the save name *)
				IF (T_Profile.T_Ctrle.sProfileName <> T_Profile.T_Id.sName) THEN
					(* overwrite the profilname with the name wrote in the file *)
					T_NovRam.T_Parameter.T_StationWork[gciStationSt1].T_InfoProcess.sProfileName:=T_Profile.T_Ctrle.sProfileName;
					T_Profile.T_IDProfileStation[T_NovRam.T_Parameter.T_StationWork[gciStationSt1].T_InfoProcess.iProfile].sName:=T_Profile.T_Ctrle.sProfileName;
					xWrongProfilNameReadedSt1:=TRUE;
				END_IF;
				(* next step *)
				iStepAction:=90;
			END_IF
			IF T_Profile.T_Ctrle.xErr THEN
				iToLoadProfileNrSt1:=T_Profile.T_Id.iNumber;
				sToLoadProfileNameSt1:=T_Profile.T_Id.sName;
				IF (T_Profile.T_Ctrle.udiErrorID <> 16#F2000) THEN
					(* Profile file not founded *)
					xProfileFileNotFoundSt1:=TRUE;
				ELSE
					(* wrong syntax of readed Profile file *)
					xProfileFileWrongSyntaxSt1:=TRUE;
				END_IF;
				(* activ reset *)
				T_Profile.T_Ctrle.xReset:=TRUE;
				(* next step *)
				iStepAction:=25;
			END_IF
		(* waiting flag *)
		25:	IF NOT T_Profile.T_Ctrle.xReset AND T_Profile.T_Ctrle.xDone THEN
				IF (T_Profile.T_Id.iNumber = 1) THEN
					T_Profile.T_LoadProfileParameter:=T_Profile.T_DefaultProfileParameter;
					T_ExchgParam.T_StationCommon.T_Param_StationWork.T_InfoProcess.iProfile:=1;
					T_ExchgParam.T_StationCommon.T_Param_StationWork.T_InfoProcess.sProfileName:='Default';
					(* erase name *)
					T_Profile.T_IDProfileStation[1].sName:='Default';
					T_NovRam.T_Parameter.T_StationWork[gciStationSt1].T_InfoProcess.iProfile:=1;
					T_NovRam.T_Parameter.T_StationWork[gciStationSt1].T_InfoProcess.sProfileName:='Default';
					iStepAction:=90;
				ELSE
					(* erase name *)
					T_Profile.T_IDProfileStation[1].sName:='Default';
					T_NovRam.T_Parameter.T_StationWork[gciStationSt1].T_InfoProcess.iProfile:=1;
					T_NovRam.T_Parameter.T_StationWork[gciStationSt1].T_InfoProcess.sProfileName:='Default';
					iStepAction:=26;
				END_IF;
			END_IF
		(* activ reading profile file *)
		26:	T_Profile.T_Ctrle.sPathAndFileName:='PROFILE\';
			T_Profile.T_Id.iNumber:=1;
			T_Profile.T_Id.sName:='Default';
			T_Profile.T_Ctrle.iFunction:=4;	(* read the profile file *)
			T_Profile.T_Ctrle.xExecute:=TRUE;
			(* next step *)
			iStepAction:=20;
		(* End function *)
		90:	xTmp:=	xProfileFileNotFoundSt1 OR xWrongProfilNameReadedSt1 OR 	xProfileFileWrongSyntaxSt1 OR xProfileFileWrongSyntax;
			IF xTmp THEN
				IF xProfileFileNotFoundSt1 THEN
					T_ExchgParam.T_SafetyCtrl.diSetForceErrorNr:=(gciStationSt1 * 1000000) + 16#F301;	(* Datei für zu ladendes Profil nicht gefunden *)
				ELSE
					IF xWrongProfilNameReadedSt1 THEN
						T_ExchgParam.T_SafetyCtrl.diSetForceErrorNr:=(gciStationSt1 * 1000000) + 16#F303;	(* Profilname von Datei ist anders als geladenes Profil *)
					END_IF;
					IF xProfileFileWrongSyntaxSt1 THEN
						T_ExchgParam.T_SafetyCtrl.diSetForceErrorNr:=(gciStationSt1 * 1000000) + 16#F304;	(* Syntaxfehler von zu ladendes Profil *)
					END_IF;
					IF xProfileFileWrongSyntax THEN
						T_ExchgParam.T_SafetyCtrl.diSetForceErrorNr:=16#F303;	(* Syntaxfehler mindestens einer Profildatei beim lesen aller Profile *)
					END_IF;
				END_IF;
				T_ExchgParam.T_SafetyCtrl.xSetForceError:=TRUE;
				xProfileFileNotFoundSt1:=xWrongProfilNameReadedSt1:=xProfileFileWrongSyntaxSt1:=FALSE;
				xProfileFileWrongSyntax:=FALSE;
			END_IF;
			T_Visu.T_CtrleAction.xDone:=TRUE;
			T_Visu.T_CtrleAction.xErr:=FALSE;
			T_Visu.T_CtrleAction.udiErrorID:=16#0;
			xAction_CopyProfileToProcess:=FALSE;
			xUpdateProfileList:=TRUE;
		(* USB-Stick is missing  *)
		98:	T_Visu.T_CtrleAction.xDone:=TRUE;
			T_Visu.T_CtrleAction.xNotReady:=FALSE;
			T_Profile.T_Ctrle.xReset:=T_Profile.T_Ctrle.xErr;
			T_ExchgParam.T_SafetyCtrl.xSetForceError:=TRUE;
			T_ExchgParam.T_SafetyCtrl.diSetForceErrorNr:=16#F300;	(* USB-Stick konnte nicht gefunden werden für Profil lesen/schreiben *)
			T_Visu.T_CtrleAction.xErr:=FALSE;
			T_Visu.T_CtrleAction.udiErrorID:=0;
			xAction_CopyProfileToProcess:=FALSE;
		END_CASE
	END_IF

